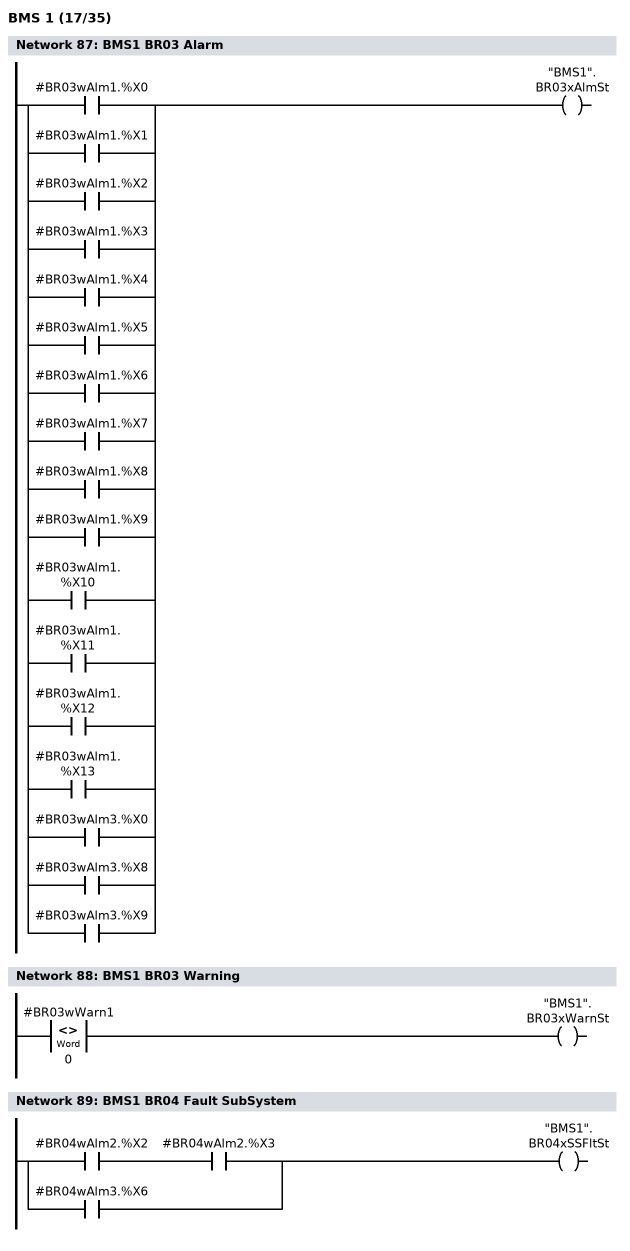
   RUNG wire#powerrail
      Contact( #BR03wAlm1.%X0 )
      wire#w1
      Coil( "BMS1".BR03xAlmSt )
   END_RUNG
   RUNG wire#powerrail
      Contact( #BR03wAlm1.%X1 )
   END_RUNG wire#w1
   RUNG wire#powerrail
      Contact( #BR03wAlm1.%X2 )
   END_RUNG wire#w1
   RUNG wire#powerrail
      Contact( #BR03wAlm1.%X3 )
   END_RUNG wire#w1
   RUNG wire#powerrail
      Contact( #BR03wAlm1.%X4 )
   END_RUNG wire#w1
   RUNG wire#powerrail
      Contact( #BR03wAlm1.%X5 )
   END_RUNG wire#w1
   RUNG wire#powerrail
      Contact( #BR03wAlm1.%X6 )
   END_RUNG wire#w1
   RUNG wire#powerrail
      Contact( #BR03wAlm1.%X7 )
   END_RUNG wire#w1
   RUNG wire#powerrail
      Contact( #BR03wAlm1.%X8 )
   END_RUNG wire#w1
   RUNG wire#powerrail
      Contact( #BR03wAlm1.%X9 )
   END_RUNG wire#w1
   RUNG wire#powerrail
      Contact( #BR03wAlm1.%X10 )
   END_RUNG wire#w1
   RUNG wire#powerrail
      Contact( #BR03wAlm1.%X11 )
   END_RUNG wire#w1
   RUNG wire#powerrail
      Contact( #BR03wAlm1.%X12 )
   END_RUNG wire#w1
   RUNG wire#powerrail
      Contact( #BR03wAlm1.%X13 )
   END_RUNG wire#w1
   RUNG wire#powerrail
      Contact( #BR03wAlm3.%X0 )
   END_RUNG wire#w1
   RUNG wire#powerrail
      Contact( #BR03wAlm3.%X8 )
   END_RUNG wire#w1
   RUNG wire#powerrail
      Contact( #BR03wAlm3.%X9 )
   END_RUNG wire#w1
   // the same network as SCL:
   "BMS1".BR03xAlmSt := #BR03wAlm1.%X0 OR #BR03wAlm1.%X1 OR #BR03wAlm1.%X2 OR #BR03wAlm1.%X3 OR #BR03wAlm1.%X4 OR #BR03wAlm1.%X5 OR #BR03wAlm1.%X6 OR #BR03wAlm1.%X7 OR #BR03wAlm1.%X8 OR #BR03wAlm1.%X9 OR #BR03wAlm1.%X10 OR #BR03wAlm1.%X11 OR #BR03wAlm1.%X12 OR #BR03wAlm1.%X13 OR #BR03wAlm3.%X0 OR #BR03wAlm3.%X8 OR #BR03wAlm3.%X9;
END_REGION

REGION Network 88: BMS1 BR03 Warning
   RUNG wire#powerrail
      { S7_Templates := "SrcType := Word" } NE_Contact(in1 := #BR03wWarn1, in2 := 0)
      Coil( "BMS1".BR03xWarnSt )
   END_RUNG
   // the same network as SCL:
   "BMS1".BR03xWarnSt := #BR03wWarn1 <> 0;
END_REGION

REGION Network 89: BMS1 BR04 Fault SubSystem
   RUNG wire#powerrail
      Contact( #BR04wAlm2.%X2 )
      Contact( #BR04wAlm2.%X3 )
      wire#w1
      Coil( "BMS1".BR04xSSFltSt )
   END_RUNG
   RUNG wire#powerrail
      Contact( #BR04wAlm3.%X6 )
   END_RUNG wire#w1
   // the same network as SCL:
   "BMS1".BR04xSSFltSt := (#BR04wAlm2.%X2 AND #BR04wAlm2.%X3) OR #BR04wAlm3.%X6;
END_REGION

REGION Network 90: BMS1 BR04 Fault
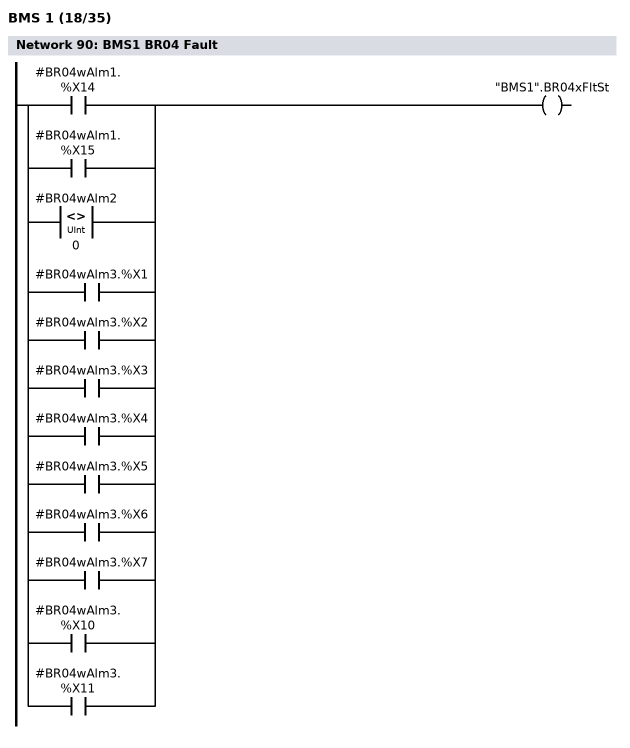
   RUNG wire#powerrail
      Contact( #BR04wAlm1.%X14 )
      wire#w1
      Coil( "BMS1".BR04xFltSt )
   END_RUNG
   RUNG wire#powerrail
      Contact( #BR04wAlm1.%X15 )
   END_RUNG wire#w1
   RUNG wire#powerrail
      { S7_Templates := "SrcType := UInt" } NE_Contact(in1 := #BR04wAlm2, in2 := 0)
   END_RUNG wire#w1
   RUNG wire#powerrail
      Contact( #BR04wAlm3.%X1 )
   END_RUNG wire#w1
   RUNG wire#powerrail
      Contact( #BR04wAlm3.%X2 )
   END_RUNG wire#w1
   RUNG wire#powerrail
      Contact( #BR04wAlm3.%X3 )
   END_RUNG wire#w1
   RUNG wire#powerrail
      Contact( #BR04wAlm3.%X4 )
   END_RUNG wire#w1
   RUNG wire#powerrail
      Contact( #BR04wAlm3.%X5 )
   END_RUNG wire#w1
   RUNG wire#powerrail
      Contact( #BR04wAlm3.%X6 )
   END_RUNG wire#w1
   RUNG wire#powerrail
      Contact( #BR04wAlm3.%X7 )
   END_RUNG wire#w1
   RUNG wire#powerrail
      Contact( #BR04wAlm3.%X10 )
   END_RUNG wire#w1
   RUNG wire#powerrail
      Contact( #BR04wAlm3.%X11 )
   END_RUNG wire#w1
   // the same network as SCL:
   "BMS1".BR04xFltSt := #BR04wAlm1.%X14 OR #BR04wAlm1.%X15 OR (#BR04wAlm2 <> 0) OR #BR04wAlm3.%X1 OR #BR04wAlm3.%X2 OR #BR04wAlm3.%X3 OR #BR04wAlm3.%X4 OR #BR04wAlm3.%X5 OR #BR04wAlm3.%X6 OR #BR04wAlm3.%X7 OR #BR04wAlm3.%X10 OR #BR04wAlm3.%X11;
END_REGION

REGION Network 91: BMS1 BR04 Alarm
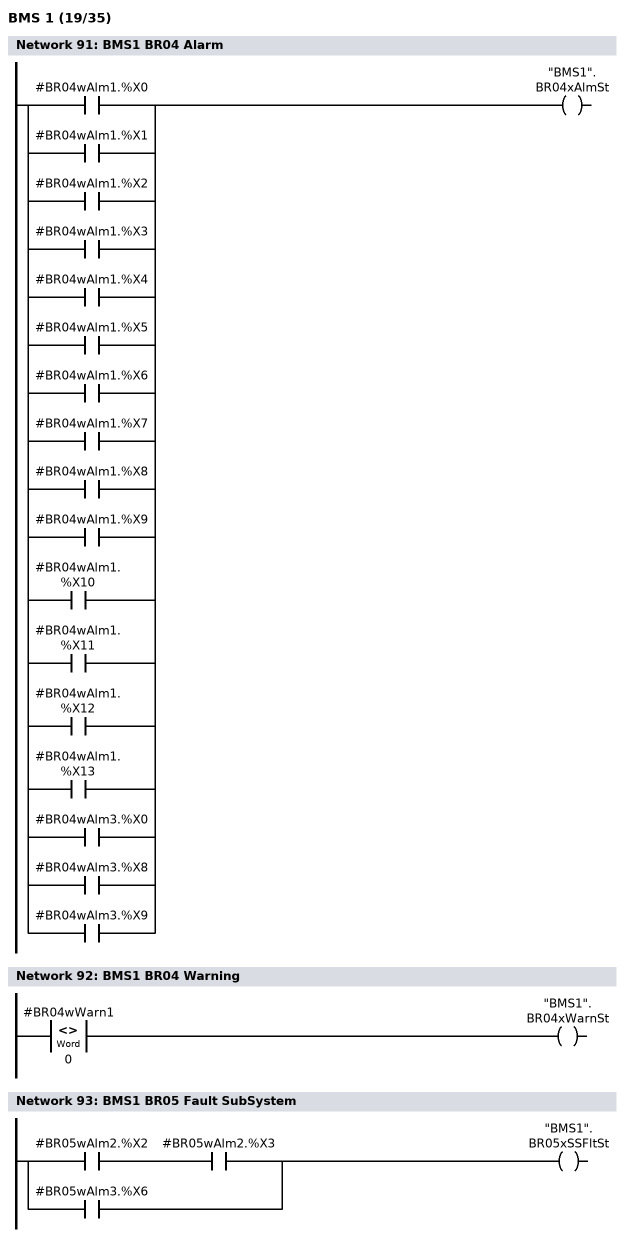
   RUNG wire#powerrail
      Contact( #BR04wAlm1.%X0 )
      wire#w1
      Coil( "BMS1".BR04xAlmSt )
   END_RUNG
   RUNG wire#powerrail
      Contact( #BR04wAlm1.%X1 )
   END_RUNG wire#w1
   RUNG wire#powerrail
      Contact( #BR04wAlm1.%X2 )
   END_RUNG wire#w1
   RUNG wire#powerrail
      Contact( #BR04wAlm1.%X3 )
   END_RUNG wire#w1
   RUNG wire#powerrail
      Contact( #BR04wAlm1.%X4 )
   END_RUNG wire#w1
   RUNG wire#powerrail
      Contact( #BR04wAlm1.%X5 )
   END_RUNG wire#w1
   RUNG wire#powerrail
      Contact( #BR04wAlm1.%X6 )
   END_RUNG wire#w1
   RUNG wire#powerrail
      Contact( #BR04wAlm1.%X7 )
   END_RUNG wire#w1
   RUNG wire#powerrail
      Contact( #BR04wAlm1.%X8 )
   END_RUNG wire#w1
   RUNG wire#powerrail
      Contact( #BR04wAlm1.%X9 )
   END_RUNG wire#w1
   RUNG wire#powerrail
      Contact( #BR04wAlm1.%X10 )
   END_RUNG wire#w1
   RUNG wire#powerrail
      Contact( #BR04wAlm1.%X11 )
   END_RUNG wire#w1
   RUNG wire#powerrail
      Contact( #BR04wAlm1.%X12 )
   END_RUNG wire#w1
   RUNG wire#powerrail
      Contact( #BR04wAlm1.%X13 )
   END_RUNG wire#w1
   RUNG wire#powerrail
      Contact( #BR04wAlm3.%X0 )
   END_RUNG wire#w1
   RUNG wire#powerrail
      Contact( #BR04wAlm3.%X8 )
   END_RUNG wire#w1
   RUNG wire#powerrail
      Contact( #BR04wAlm3.%X9 )
   END_RUNG wire#w1
   // the same network as SCL:
   "BMS1".BR04xAlmSt := #BR04wAlm1.%X0 OR #BR04wAlm1.%X1 OR #BR04wAlm1.%X2 OR #BR04wAlm1.%X3 OR #BR04wAlm1.%X4 OR #BR04wAlm1.%X5 OR #BR04wAlm1.%X6 OR #BR04wAlm1.%X7 OR #BR04wAlm1.%X8 OR #BR04wAlm1.%X9 OR #BR04wAlm1.%X10 OR #BR04wAlm1.%X11 OR #BR04wAlm1.%X12 OR #BR04wAlm1.%X13 OR #BR04wAlm3.%X0 OR #BR04wAlm3.%X8 OR #BR04wAlm3.%X9;
END_REGION

REGION Network 92: BMS1 BR04 Warning
   RUNG wire#powerrail
      { S7_Templates := "SrcType := Word" } NE_Contact(in1 := #BR04wWarn1, in2 := 0)
      Coil( "BMS1".BR04xWarnSt )
   END_RUNG
   // the same network as SCL:
   "BMS1".BR04xWarnSt := #BR04wWarn1 <> 0;
END_REGION

REGION Network 93: BMS1 BR05 Fault SubSystem
   RUNG wire#powerrail
      Contact( #BR05wAlm2.%X2 )
      Contact( #BR05wAlm2.%X3 )
      wire#w1
      Coil( "BMS1".BR05xSSFltSt )
   END_RUNG
   RUNG wire#powerrail
      Contact( #BR05wAlm3.%X6 )
   END_RUNG wire#w1
   // the same network as SCL:
   "BMS1".BR05xSSFltSt := (#BR05wAlm2.%X2 AND #BR05wAlm2.%X3) OR #BR05wAlm3.%X6;
END_REGION

REGION Network 94: BMS1 BR05 Fault
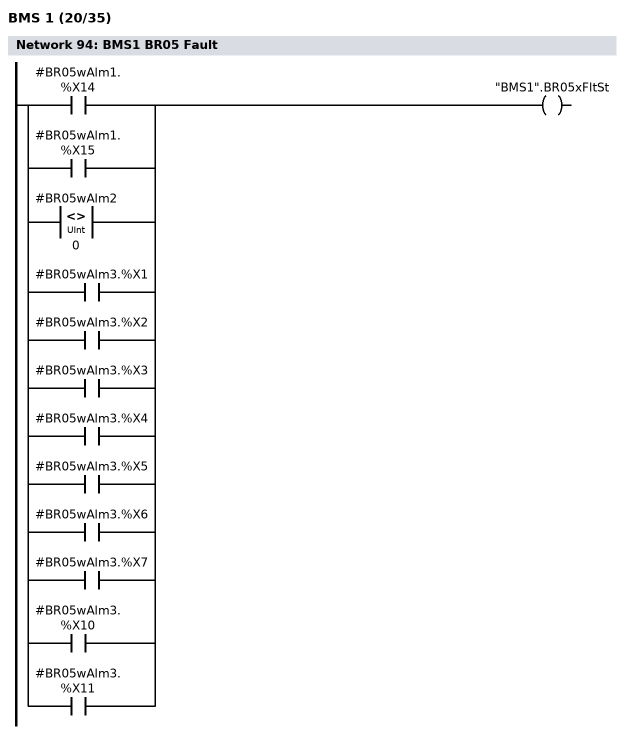
   RUNG wire#powerrail
      Contact( #BR05wAlm1.%X14 )
      wire#w1
      Coil( "BMS1".BR05xFltSt )
   END_RUNG
   RUNG wire#powerrail
      Contact( #BR05wAlm1.%X15 )
   END_RUNG wire#w1
   RUNG wire#powerrail
      { S7_Templates := "SrcType := UInt" } NE_Contact(in1 := #BR05wAlm2, in2 := 0)
   END_RUNG wire#w1
   RUNG wire#powerrail
      Contact( #BR05wAlm3.%X1 )
   END_RUNG wire#w1
   RUNG wire#powerrail
      Contact( #BR05wAlm3.%X2 )
   END_RUNG wire#w1
   RUNG wire#powerrail
      Contact( #BR05wAlm3.%X3 )
   END_RUNG wire#w1
   RUNG wire#powerrail
      Contact( #BR05wAlm3.%X4 )
   END_RUNG wire#w1
   RUNG wire#powerrail
      Contact( #BR05wAlm3.%X5 )
   END_RUNG wire#w1
   RUNG wire#powerrail
      Contact( #BR05wAlm3.%X6 )
   END_RUNG wire#w1
   RUNG wire#powerrail
      Contact( #BR05wAlm3.%X7 )
   END_RUNG wire#w1
   RUNG wire#powerrail
      Contact( #BR05wAlm3.%X10 )
   END_RUNG wire#w1
   RUNG wire#powerrail
      Contact( #BR05wAlm3.%X11 )
   END_RUNG wire#w1
   // the same network as SCL:
   "BMS1".BR05xFltSt := #BR05wAlm1.%X14 OR #BR05wAlm1.%X15 OR (#BR05wAlm2 <> 0) OR #BR05wAlm3.%X1 OR #BR05wAlm3.%X2 OR #BR05wAlm3.%X3 OR #BR05wAlm3.%X4 OR #BR05wAlm3.%X5 OR #BR05wAlm3.%X6 OR #BR05wAlm3.%X7 OR #BR05wAlm3.%X10 OR #BR05wAlm3.%X11;
END_REGION

REGION Network 95: BMS1 BR05 Alarm
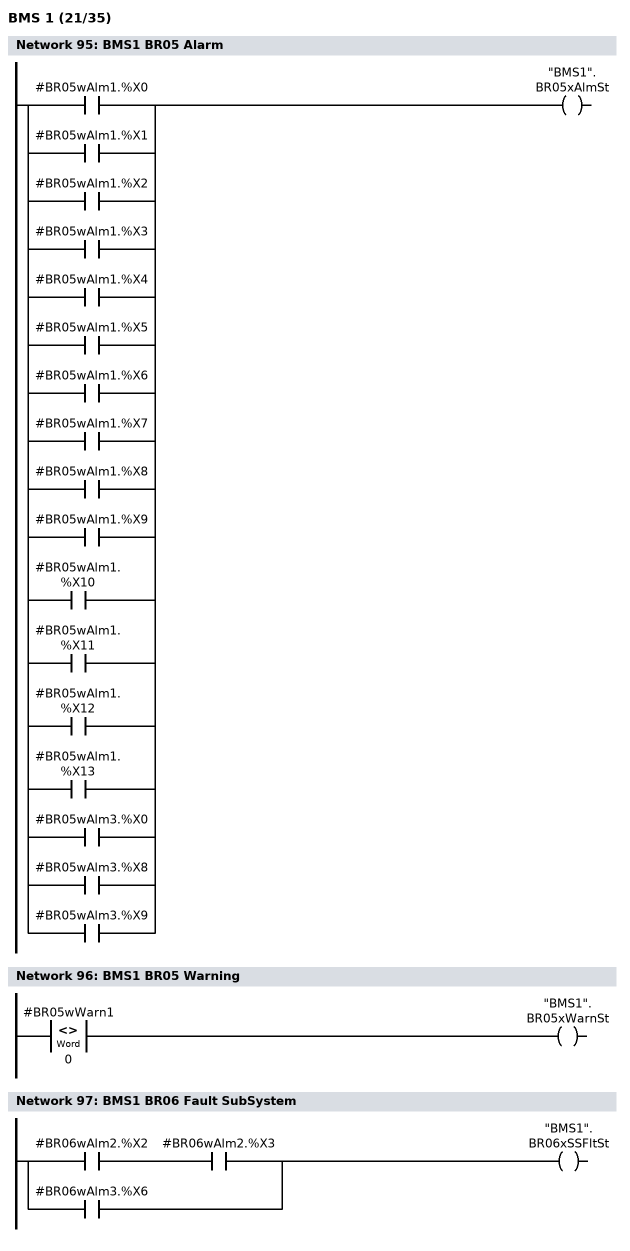
   RUNG wire#powerrail
      Contact( #BR05wAlm1.%X0 )
      wire#w1
      Coil( "BMS1".BR05xAlmSt )
   END_RUNG
   RUNG wire#powerrail
      Contact( #BR05wAlm1.%X1 )
   END_RUNG wire#w1
   RUNG wire#powerrail
      Contact( #BR05wAlm1.%X2 )
   END_RUNG wire#w1
   RUNG wire#powerrail
      Contact( #BR05wAlm1.%X3 )
   END_RUNG wire#w1
   RUNG wire#powerrail
      Contact( #BR05wAlm1.%X4 )
   END_RUNG wire#w1
   RUNG wire#powerrail
      Contact( #BR05wAlm1.%X5 )
   END_RUNG wire#w1
   RUNG wire#powerrail
      Contact( #BR05wAlm1.%X6 )
   END_RUNG wire#w1
   RUNG wire#powerrail
      Contact( #BR05wAlm1.%X7 )
   END_RUNG wire#w1
   RUNG wire#powerrail
      Contact( #BR05wAlm1.%X8 )
   END_RUNG wire#w1
   RUNG wire#powerrail
      Contact( #BR05wAlm1.%X9 )
   END_RUNG wire#w1
   RUNG wire#powerrail
      Contact( #BR05wAlm1.%X10 )
   END_RUNG wire#w1
   RUNG wire#powerrail
      Contact( #BR05wAlm1.%X11 )
   END_RUNG wire#w1
   RUNG wire#powerrail
      Contact( #BR05wAlm1.%X12 )
   END_RUNG wire#w1
   RUNG wire#powerrail
      Contact( #BR05wAlm1.%X13 )
   END_RUNG wire#w1
   RUNG wire#powerrail
      Contact( #BR05wAlm3.%X0 )
   END_RUNG wire#w1
   RUNG wire#powerrail
      Contact( #BR05wAlm3.%X8 )
   END_RUNG wire#w1
   RUNG wire#powerrail
      Contact( #BR05wAlm3.%X9 )
   END_RUNG wire#w1
   // the same network as SCL:
   "BMS1".BR05xAlmSt := #BR05wAlm1.%X0 OR #BR05wAlm1.%X1 OR #BR05wAlm1.%X2 OR #BR05wAlm1.%X3 OR #BR05wAlm1.%X4 OR #BR05wAlm1.%X5 OR #BR05wAlm1.%X6 OR #BR05wAlm1.%X7 OR #BR05wAlm1.%X8 OR #BR05wAlm1.%X9 OR #BR05wAlm1.%X10 OR #BR05wAlm1.%X11 OR #BR05wAlm1.%X12 OR #BR05wAlm1.%X13 OR #BR05wAlm3.%X0 OR #BR05wAlm3.%X8 OR #BR05wAlm3.%X9;
END_REGION

REGION Network 96: BMS1 BR05 Warning
   RUNG wire#powerrail
      { S7_Templates := "SrcType := Word" } NE_Contact(in1 := #BR05wWarn1, in2 := 0)
      Coil( "BMS1".BR05xWarnSt )
   END_RUNG
   // the same network as SCL:
   "BMS1".BR05xWarnSt := #BR05wWarn1 <> 0;
END_REGION

REGION Network 97: BMS1 BR06 Fault SubSystem
   RUNG wire#powerrail
      Contact( #BR06wAlm2.%X2 )
      Contact( #BR06wAlm2.%X3 )
      wire#w1
      Coil( "BMS1".BR06xSSFltSt )
   END_RUNG
   RUNG wire#powerrail
      Contact( #BR06wAlm3.%X6 )
   END_RUNG wire#w1
   // the same network as SCL:
   "BMS1".BR06xSSFltSt := (#BR06wAlm2.%X2 AND #BR06wAlm2.%X3) OR #BR06wAlm3.%X6;
END_REGION

REGION Network 98: BMS1 BR06 Fault
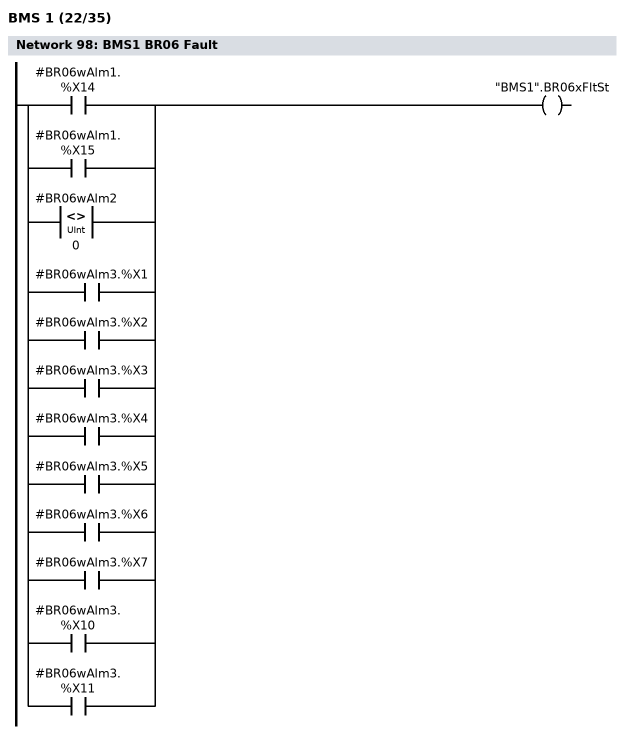
   RUNG wire#powerrail
      Contact( #BR06wAlm1.%X14 )
      wire#w1
      Coil( "BMS1".BR06xFltSt )
   END_RUNG
   RUNG wire#powerrail
      Contact( #BR06wAlm1.%X15 )
   END_RUNG wire#w1
   RUNG wire#powerrail
      { S7_Templates := "SrcType := UInt" } NE_Contact(in1 := #BR06wAlm2, in2 := 0)
   END_RUNG wire#w1
   RUNG wire#powerrail
      Contact( #BR06wAlm3.%X1 )
   END_RUNG wire#w1
   RUNG wire#powerrail
      Contact( #BR06wAlm3.%X2 )
   END_RUNG wire#w1
   RUNG wire#powerrail
      Contact( #BR06wAlm3.%X3 )
   END_RUNG wire#w1
   RUNG wire#powerrail
      Contact( #BR06wAlm3.%X4 )
   END_RUNG wire#w1
   RUNG wire#powerrail
      Contact( #BR06wAlm3.%X5 )
   END_RUNG wire#w1
   RUNG wire#powerrail
      Contact( #BR06wAlm3.%X6 )
   END_RUNG wire#w1
   RUNG wire#powerrail
      Contact( #BR06wAlm3.%X7 )
   END_RUNG wire#w1
   RUNG wire#powerrail
      Contact( #BR06wAlm3.%X10 )
   END_RUNG wire#w1
   RUNG wire#powerrail
      Contact( #BR06wAlm3.%X11 )
   END_RUNG wire#w1
   // the same network as SCL:
   "BMS1".BR06xFltSt := #BR06wAlm1.%X14 OR #BR06wAlm1.%X15 OR (#BR06wAlm2 <> 0) OR #BR06wAlm3.%X1 OR #BR06wAlm3.%X2 OR #BR06wAlm3.%X3 OR #BR06wAlm3.%X4 OR #BR06wAlm3.%X5 OR #BR06wAlm3.%X6 OR #BR06wAlm3.%X7 OR #BR06wAlm3.%X10 OR #BR06wAlm3.%X11;
END_REGION

REGION Network 99: BMS1 BR06 Alarm
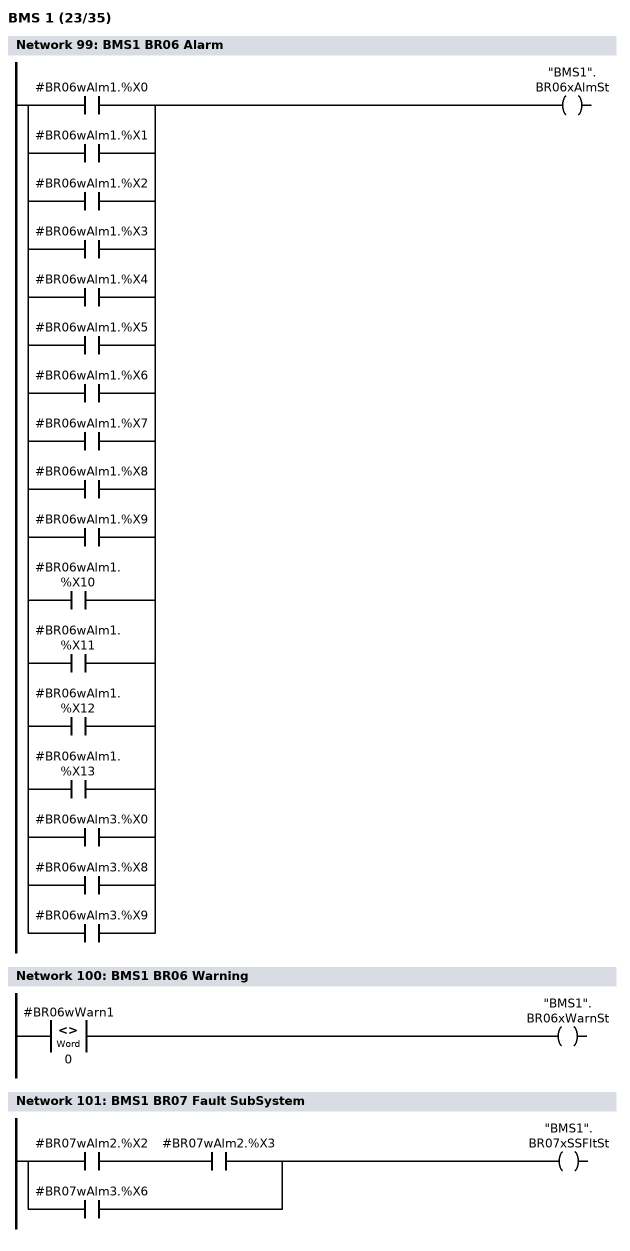
   RUNG wire#powerrail
      Contact( #BR06wAlm1.%X0 )
      wire#w1
      Coil( "BMS1".BR06xAlmSt )
   END_RUNG
   RUNG wire#powerrail
      Contact( #BR06wAlm1.%X1 )
   END_RUNG wire#w1
   RUNG wire#powerrail
      Contact( #BR06wAlm1.%X2 )
   END_RUNG wire#w1
   RUNG wire#powerrail
      Contact( #BR06wAlm1.%X3 )
   END_RUNG wire#w1
   RUNG wire#powerrail
      Contact( #BR06wAlm1.%X4 )
   END_RUNG wire#w1
   RUNG wire#powerrail
      Contact( #BR06wAlm1.%X5 )
   END_RUNG wire#w1
   RUNG wire#powerrail
      Contact( #BR06wAlm1.%X6 )
   END_RUNG wire#w1
   RUNG wire#powerrail
      Contact( #BR06wAlm1.%X7 )
   END_RUNG wire#w1
   RUNG wire#powerrail
      Contact( #BR06wAlm1.%X8 )
   END_RUNG wire#w1
   RUNG wire#powerrail
      Contact( #BR06wAlm1.%X9 )
   END_RUNG wire#w1
   RUNG wire#powerrail
      Contact( #BR06wAlm1.%X10 )
   END_RUNG wire#w1
   RUNG wire#powerrail
      Contact( #BR06wAlm1.%X11 )
   END_RUNG wire#w1
   RUNG wire#powerrail
      Contact( #BR06wAlm1.%X12 )
   END_RUNG wire#w1
   RUNG wire#powerrail
      Contact( #BR06wAlm1.%X13 )
   END_RUNG wire#w1
   RUNG wire#powerrail
      Contact( #BR06wAlm3.%X0 )
   END_RUNG wire#w1
   RUNG wire#powerrail
      Contact( #BR06wAlm3.%X8 )
   END_RUNG wire#w1
   RUNG wire#powerrail
      Contact( #BR06wAlm3.%X9 )
   END_RUNG wire#w1
   // the same network as SCL:
   "BMS1".BR06xAlmSt := #BR06wAlm1.%X0 OR #BR06wAlm1.%X1 OR #BR06wAlm1.%X2 OR #BR06wAlm1.%X3 OR #BR06wAlm1.%X4 OR #BR06wAlm1.%X5 OR #BR06wAlm1.%X6 OR #BR06wAlm1.%X7 OR #BR06wAlm1.%X8 OR #BR06wAlm1.%X9 OR #BR06wAlm1.%X10 OR #BR06wAlm1.%X11 OR #BR06wAlm1.%X12 OR #BR06wAlm1.%X13 OR #BR06wAlm3.%X0 OR #BR06wAlm3.%X8 OR #BR06wAlm3.%X9;
END_REGION

REGION Network 100: BMS1 BR06 Warning
   RUNG wire#powerrail
      { S7_Templates := "SrcType := Word" } NE_Contact(in1 := #BR06wWarn1, in2 := 0)
      Coil( "BMS1".BR06xWarnSt )
   END_RUNG
   // the same network as SCL:
   "BMS1".BR06xWarnSt := #BR06wWarn1 <> 0;
END_REGION

REGION Network 101: BMS1 BR07 Fault SubSystem
   RUNG wire#powerrail
      Contact( #BR07wAlm2.%X2 )
      Contact( #BR07wAlm2.%X3 )
      wire#w1
      Coil( "BMS1".BR07xSSFltSt )
   END_RUNG
   RUNG wire#powerrail
      Contact( #BR07wAlm3.%X6 )
   END_RUNG wire#w1
   // the same network as SCL:
   "BMS1".BR07xSSFltSt := (#BR07wAlm2.%X2 AND #BR07wAlm2.%X3) OR #BR07wAlm3.%X6;
END_REGION

REGION Network 102: BMS1 BR07 Fault
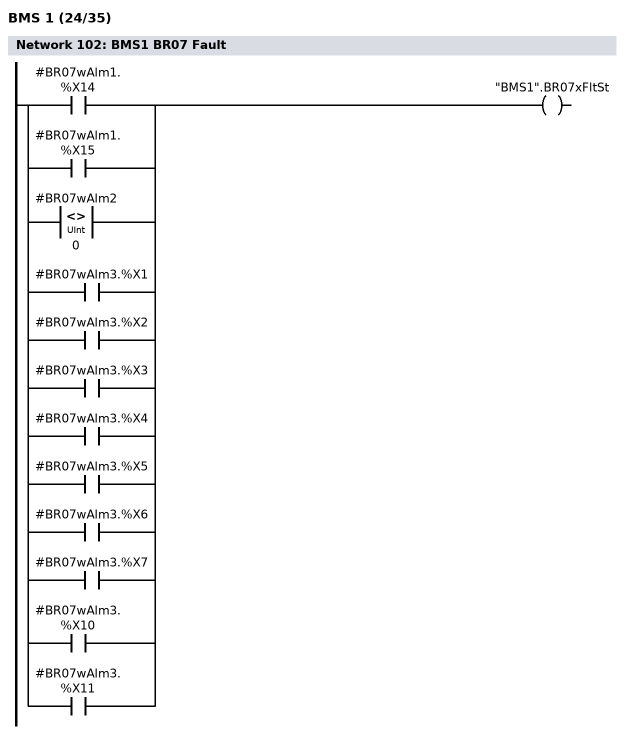
   RUNG wire#powerrail
      Contact( #BR07wAlm1.%X14 )
      wire#w1
      Coil( "BMS1".BR07xFltSt )
   END_RUNG
   RUNG wire#powerrail
      Contact( #BR07wAlm1.%X15 )
   END_RUNG wire#w1
   RUNG wire#powerrail
      { S7_Templates := "SrcType := UInt" } NE_Contact(in1 := #BR07wAlm2, in2 := 0)
   END_RUNG wire#w1
   RUNG wire#powerrail
      Contact( #BR07wAlm3.%X1 )
   END_RUNG wire#w1
   RUNG wire#powerrail
      Contact( #BR07wAlm3.%X2 )
   END_RUNG wire#w1
   RUNG wire#powerrail
      Contact( #BR07wAlm3.%X3 )
   END_RUNG wire#w1
   RUNG wire#powerrail
      Contact( #BR07wAlm3.%X4 )
   END_RUNG wire#w1
   RUNG wire#powerrail
      Contact( #BR07wAlm3.%X5 )
   END_RUNG wire#w1
   RUNG wire#powerrail
      Contact( #BR07wAlm3.%X6 )
   END_RUNG wire#w1
   RUNG wire#powerrail
      Contact( #BR07wAlm3.%X7 )
   END_RUNG wire#w1
   RUNG wire#powerrail
      Contact( #BR07wAlm3.%X10 )
   END_RUNG wire#w1
   RUNG wire#powerrail
      Contact( #BR07wAlm3.%X11 )
   END_RUNG wire#w1
   // the same network as SCL:
   "BMS1".BR07xFltSt := #BR07wAlm1.%X14 OR #BR07wAlm1.%X15 OR (#BR07wAlm2 <> 0) OR #BR07wAlm3.%X1 OR #BR07wAlm3.%X2 OR #BR07wAlm3.%X3 OR #BR07wAlm3.%X4 OR #BR07wAlm3.%X5 OR #BR07wAlm3.%X6 OR #BR07wAlm3.%X7 OR #BR07wAlm3.%X10 OR #BR07wAlm3.%X11;
END_REGION

REGION Network 103: BMS1 BR07 Alarm
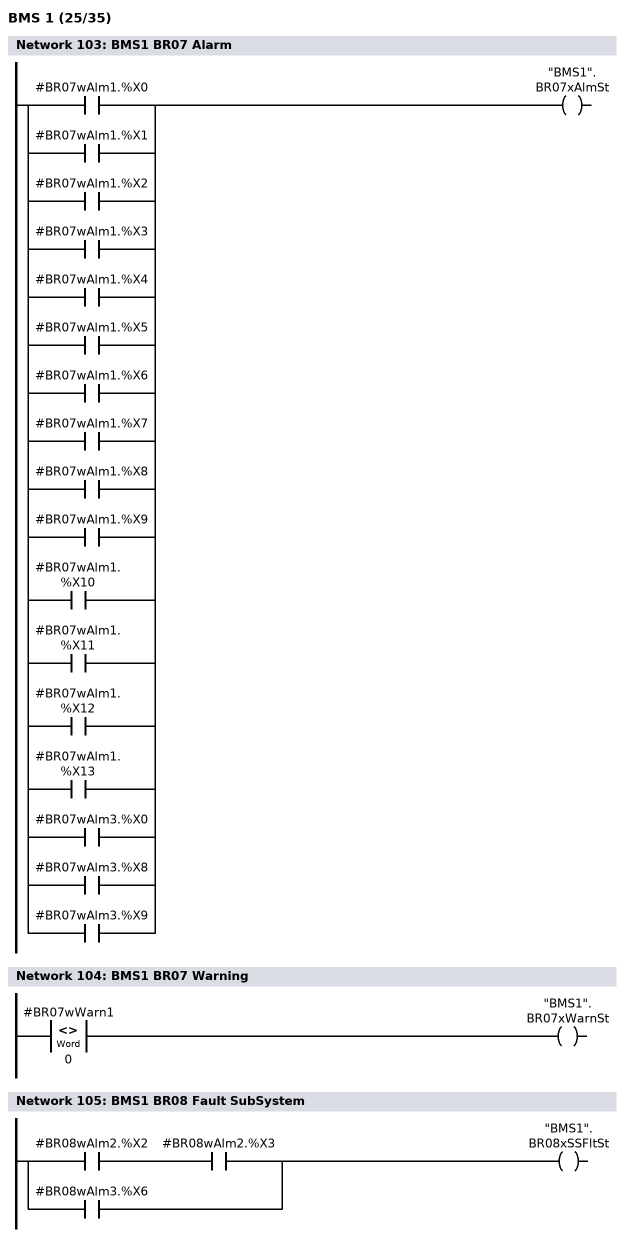
   RUNG wire#powerrail
      Contact( #BR07wAlm1.%X0 )
      wire#w1
      Coil( "BMS1".BR07xAlmSt )
   END_RUNG
   RUNG wire#powerrail
      Contact( #BR07wAlm1.%X1 )
   END_RUNG wire#w1
   RUNG wire#powerrail
      Contact( #BR07wAlm1.%X2 )
   END_RUNG wire#w1
   RUNG wire#powerrail
      Contact( #BR07wAlm1.%X3 )
   END_RUNG wire#w1
   RUNG wire#powerrail
      Contact( #BR07wAlm1.%X4 )
   END_RUNG wire#w1
   RUNG wire#powerrail
      Contact( #BR07wAlm1.%X5 )
   END_RUNG wire#w1
   RUNG wire#powerrail
      Contact( #BR07wAlm1.%X6 )
   END_RUNG wire#w1
   RUNG wire#powerrail
      Contact( #BR07wAlm1.%X7 )
   END_RUNG wire#w1
   RUNG wire#powerrail
      Contact( #BR07wAlm1.%X8 )
   END_RUNG wire#w1
   RUNG wire#powerrail
      Contact( #BR07wAlm1.%X9 )
   END_RUNG wire#w1
   RUNG wire#powerrail
      Contact( #BR07wAlm1.%X10 )
   END_RUNG wire#w1
   RUNG wire#powerrail
      Contact( #BR07wAlm1.%X11 )
   END_RUNG wire#w1
   RUNG wire#powerrail
      Contact( #BR07wAlm1.%X12 )
   END_RUNG wire#w1
   RUNG wire#powerrail
      Contact( #BR07wAlm1.%X13 )
   END_RUNG wire#w1
   RUNG wire#powerrail
      Contact( #BR07wAlm3.%X0 )
   END_RUNG wire#w1
   RUNG wire#powerrail
      Contact( #BR07wAlm3.%X8 )
   END_RUNG wire#w1
   RUNG wire#powerrail
      Contact( #BR07wAlm3.%X9 )
   END_RUNG wire#w1
   // the same network as SCL:
   "BMS1".BR07xAlmSt := #BR07wAlm1.%X0 OR #BR07wAlm1.%X1 OR #BR07wAlm1.%X2 OR #BR07wAlm1.%X3 OR #BR07wAlm1.%X4 OR #BR07wAlm1.%X5 OR #BR07wAlm1.%X6 OR #BR07wAlm1.%X7 OR #BR07wAlm1.%X8 OR #BR07wAlm1.%X9 OR #BR07wAlm1.%X10 OR #BR07wAlm1.%X11 OR #BR07wAlm1.%X12 OR #BR07wAlm1.%X13 OR #BR07wAlm3.%X0 OR #BR07wAlm3.%X8 OR #BR07wAlm3.%X9;
END_REGION

REGION Network 104: BMS1 BR07 Warning
   RUNG wire#powerrail
      { S7_Templates := "SrcType := Word" } NE_Contact(in1 := #BR07wWarn1, in2 := 0)
      Coil( "BMS1".BR07xWarnSt )
   END_RUNG
   // the same network as SCL:
   "BMS1".BR07xWarnSt := #BR07wWarn1 <> 0;
END_REGION

REGION Network 105: BMS1 BR08 Fault SubSystem
   RUNG wire#powerrail
      Contact( #BR08wAlm2.%X2 )
      Contact( #BR08wAlm2.%X3 )
      wire#w1
      Coil( "BMS1".BR08xSSFltSt )
   END_RUNG
   RUNG wire#powerrail
      Contact( #BR08wAlm3.%X6 )
   END_RUNG wire#w1
   // the same network as SCL:
   "BMS1".BR08xSSFltSt := (#BR08wAlm2.%X2 AND #BR08wAlm2.%X3) OR #BR08wAlm3.%X6;
END_REGION

REGION Network 106: BMS1 BR08 Fault
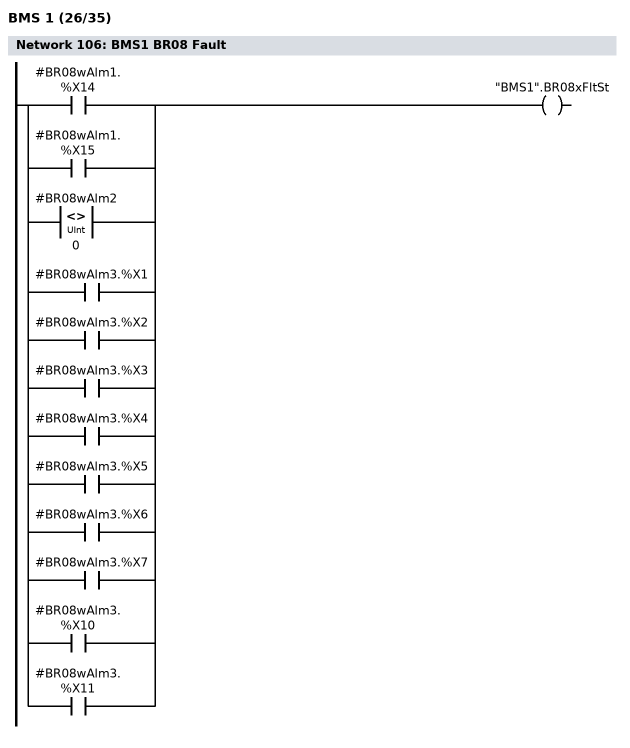
   RUNG wire#powerrail
      Contact( #BR08wAlm1.%X14 )
      wire#w1
      Coil( "BMS1".BR08xFltSt )
   END_RUNG
   RUNG wire#powerrail
      Contact( #BR08wAlm1.%X15 )
   END_RUNG wire#w1
   RUNG wire#powerrail
      { S7_Templates := "SrcType := UInt" } NE_Contact(in1 := #BR08wAlm2, in2 := 0)
   END_RUNG wire#w1
   RUNG wire#powerrail
      Contact( #BR08wAlm3.%X1 )
   END_RUNG wire#w1
   RUNG wire#powerrail
      Contact( #BR08wAlm3.%X2 )
   END_RUNG wire#w1
   RUNG wire#powerrail
      Contact( #BR08wAlm3.%X3 )
   END_RUNG wire#w1
   RUNG wire#powerrail
      Contact( #BR08wAlm3.%X4 )
   END_RUNG wire#w1
   RUNG wire#powerrail
      Contact( #BR08wAlm3.%X5 )
   END_RUNG wire#w1
   RUNG wire#powerrail
      Contact( #BR08wAlm3.%X6 )
   END_RUNG wire#w1
   RUNG wire#powerrail
      Contact( #BR08wAlm3.%X7 )
   END_RUNG wire#w1
   RUNG wire#powerrail
      Contact( #BR08wAlm3.%X10 )
   END_RUNG wire#w1
   RUNG wire#powerrail
      Contact( #BR08wAlm3.%X11 )
   END_RUNG wire#w1
   // the same network as SCL:
   "BMS1".BR08xFltSt := #BR08wAlm1.%X14 OR #BR08wAlm1.%X15 OR (#BR08wAlm2 <> 0) OR #BR08wAlm3.%X1 OR #BR08wAlm3.%X2 OR #BR08wAlm3.%X3 OR #BR08wAlm3.%X4 OR #BR08wAlm3.%X5 OR #BR08wAlm3.%X6 OR #BR08wAlm3.%X7 OR #BR08wAlm3.%X10 OR #BR08wAlm3.%X11;
END_REGION

REGION Network 107: BMS1 BR08 Alarm
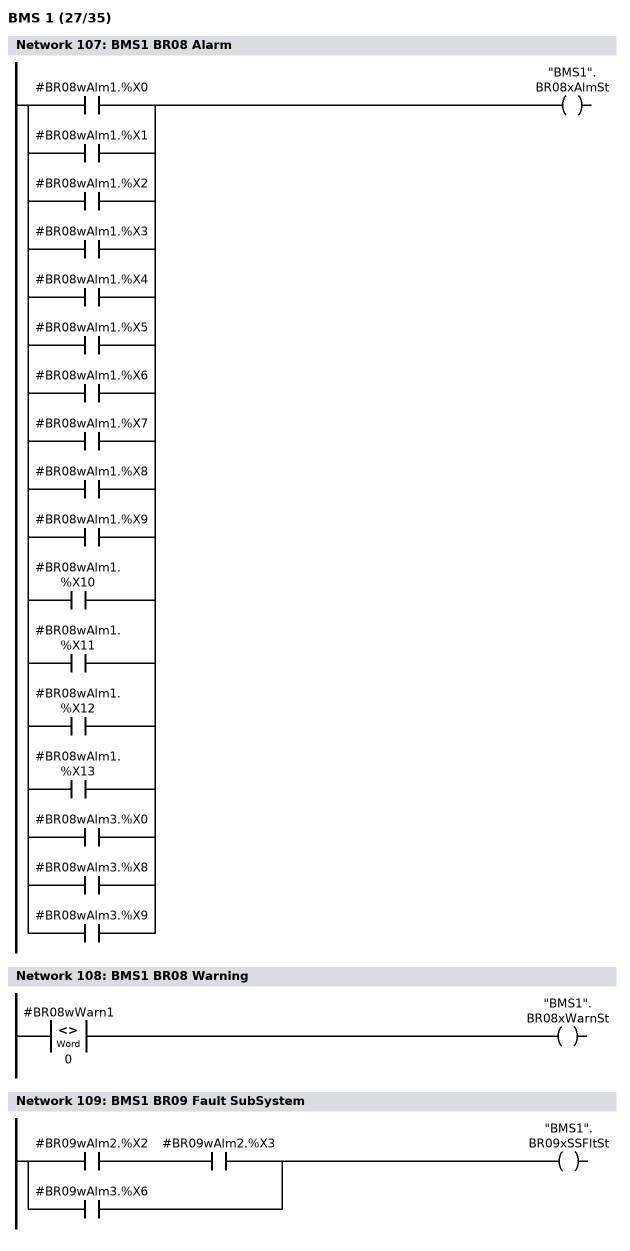
   RUNG wire#powerrail
      Contact( #BR08wAlm1.%X0 )
      wire#w1
      Coil( "BMS1".BR08xAlmSt )
   END_RUNG
   RUNG wire#powerrail
      Contact( #BR08wAlm1.%X1 )
   END_RUNG wire#w1
   RUNG wire#powerrail
      Contact( #BR08wAlm1.%X2 )
   END_RUNG wire#w1
   RUNG wire#powerrail
      Contact( #BR08wAlm1.%X3 )
   END_RUNG wire#w1
   RUNG wire#powerrail
      Contact( #BR08wAlm1.%X4 )
   END_RUNG wire#w1
   RUNG wire#powerrail
      Contact( #BR08wAlm1.%X5 )
   END_RUNG wire#w1
   RUNG wire#powerrail
      Contact( #BR08wAlm1.%X6 )
   END_RUNG wire#w1
   RUNG wire#powerrail
      Contact( #BR08wAlm1.%X7 )
   END_RUNG wire#w1
   RUNG wire#powerrail
      Contact( #BR08wAlm1.%X8 )
   END_RUNG wire#w1
   RUNG wire#powerrail
      Contact( #BR08wAlm1.%X9 )
   END_RUNG wire#w1
   RUNG wire#powerrail
      Contact( #BR08wAlm1.%X10 )
   END_RUNG wire#w1
   RUNG wire#powerrail
      Contact( #BR08wAlm1.%X11 )
   END_RUNG wire#w1
   RUNG wire#powerrail
      Contact( #BR08wAlm1.%X12 )
   END_RUNG wire#w1
   RUNG wire#powerrail
      Contact( #BR08wAlm1.%X13 )
   END_RUNG wire#w1
   RUNG wire#powerrail
      Contact( #BR08wAlm3.%X0 )
   END_RUNG wire#w1
   RUNG wire#powerrail
      Contact( #BR08wAlm3.%X8 )
   END_RUNG wire#w1
   RUNG wire#powerrail
      Contact( #BR08wAlm3.%X9 )
   END_RUNG wire#w1
   // the same network as SCL:
   "BMS1".BR08xAlmSt := #BR08wAlm1.%X0 OR #BR08wAlm1.%X1 OR #BR08wAlm1.%X2 OR #BR08wAlm1.%X3 OR #BR08wAlm1.%X4 OR #BR08wAlm1.%X5 OR #BR08wAlm1.%X6 OR #BR08wAlm1.%X7 OR #BR08wAlm1.%X8 OR #BR08wAlm1.%X9 OR #BR08wAlm1.%X10 OR #BR08wAlm1.%X11 OR #BR08wAlm1.%X12 OR #BR08wAlm1.%X13 OR #BR08wAlm3.%X0 OR #BR08wAlm3.%X8 OR #BR08wAlm3.%X9;
END_REGION

REGION Network 108: BMS1 BR08 Warning
   RUNG wire#powerrail
      { S7_Templates := "SrcType := Word" } NE_Contact(in1 := #BR08wWarn1, in2 := 0)
      Coil( "BMS1".BR08xWarnSt )
   END_RUNG
   // the same network as SCL:
   "BMS1".BR08xWarnSt := #BR08wWarn1 <> 0;
END_REGION

REGION Network 109: BMS1 BR09 Fault SubSystem
   RUNG wire#powerrail
      Contact( #BR09wAlm2.%X2 )
      Contact( #BR09wAlm2.%X3 )
      wire#w1
      Coil( "BMS1".BR09xSSFltSt )
   END_RUNG
   RUNG wire#powerrail
      Contact( #BR09wAlm3.%X6 )
   END_RUNG wire#w1
   // the same network as SCL:
   "BMS1".BR09xSSFltSt := (#BR09wAlm2.%X2 AND #BR09wAlm2.%X3) OR #BR09wAlm3.%X6;
END_REGION

REGION Network 110: BMS1 BR09 Fault
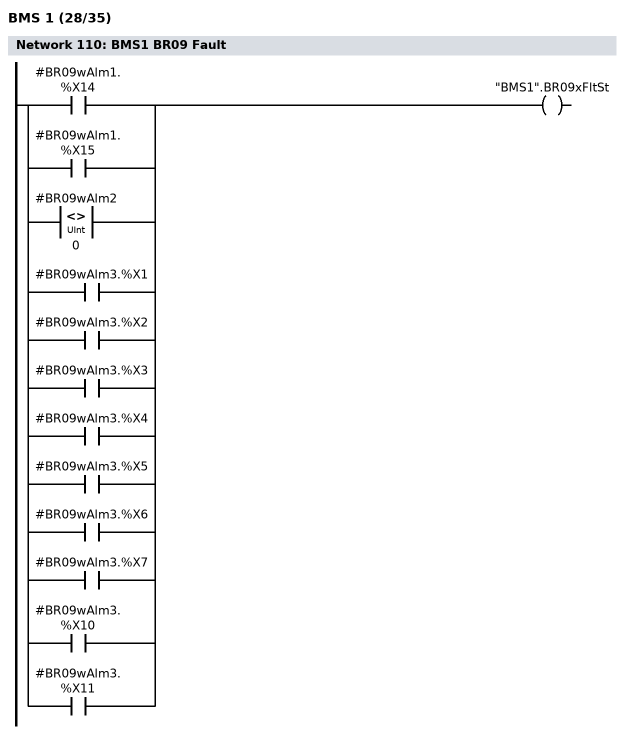
   RUNG wire#powerrail
      Contact( #BR09wAlm1.%X14 )
      wire#w1
      Coil( "BMS1".BR09xFltSt )
   END_RUNG
   RUNG wire#powerrail
      Contact( #BR09wAlm1.%X15 )
   END_RUNG wire#w1
   RUNG wire#powerrail
      { S7_Templates := "SrcType := UInt" } NE_Contact(in1 := #BR09wAlm2, in2 := 0)
   END_RUNG wire#w1
   RUNG wire#powerrail
      Contact( #BR09wAlm3.%X1 )
   END_RUNG wire#w1
   RUNG wire#powerrail
      Contact( #BR09wAlm3.%X2 )
   END_RUNG wire#w1
   RUNG wire#powerrail
      Contact( #BR09wAlm3.%X3 )
   END_RUNG wire#w1
   RUNG wire#powerrail
      Contact( #BR09wAlm3.%X4 )
   END_RUNG wire#w1
   RUNG wire#powerrail
      Contact( #BR09wAlm3.%X5 )
   END_RUNG wire#w1
   RUNG wire#powerrail
      Contact( #BR09wAlm3.%X6 )
   END_RUNG wire#w1
   RUNG wire#powerrail
      Contact( #BR09wAlm3.%X7 )
   END_RUNG wire#w1
   RUNG wire#powerrail
      Contact( #BR09wAlm3.%X10 )
   END_RUNG wire#w1
   RUNG wire#powerrail
      Contact( #BR09wAlm3.%X11 )
   END_RUNG wire#w1
   // the same network as SCL:
   "BMS1".BR09xFltSt := #BR09wAlm1.%X14 OR #BR09wAlm1.%X15 OR (#BR09wAlm2 <> 0) OR #BR09wAlm3.%X1 OR #BR09wAlm3.%X2 OR #BR09wAlm3.%X3 OR #BR09wAlm3.%X4 OR #BR09wAlm3.%X5 OR #BR09wAlm3.%X6 OR #BR09wAlm3.%X7 OR #BR09wAlm3.%X10 OR #BR09wAlm3.%X11;
END_REGION

REGION Network 111: BMS1 BR09 Alarm
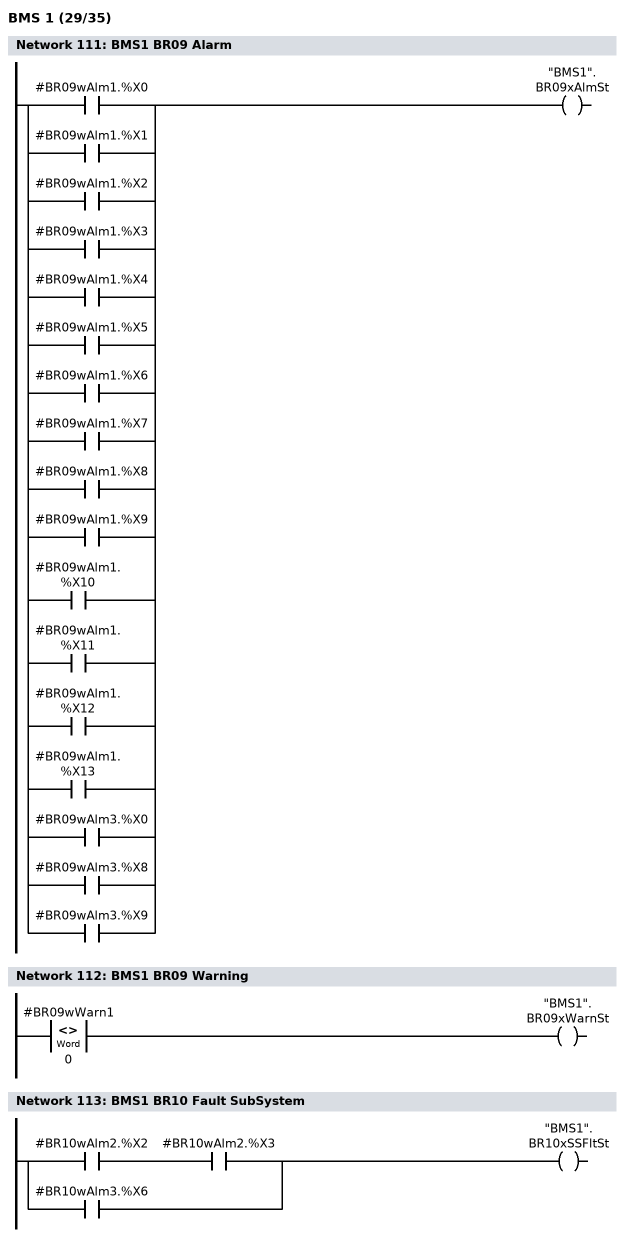
   RUNG wire#powerrail
      Contact( #BR09wAlm1.%X0 )
      wire#w1
      Coil( "BMS1".BR09xAlmSt )
   END_RUNG
   RUNG wire#powerrail
      Contact( #BR09wAlm1.%X1 )
   END_RUNG wire#w1
   RUNG wire#powerrail
      Contact( #BR09wAlm1.%X2 )
   END_RUNG wire#w1
   RUNG wire#powerrail
      Contact( #BR09wAlm1.%X3 )
   END_RUNG wire#w1
   RUNG wire#powerrail
      Contact( #BR09wAlm1.%X4 )
   END_RUNG wire#w1
   RUNG wire#powerrail
      Contact( #BR09wAlm1.%X5 )
   END_RUNG wire#w1
   RUNG wire#powerrail
      Contact( #BR09wAlm1.%X6 )
   END_RUNG wire#w1
   RUNG wire#powerrail
      Contact( #BR09wAlm1.%X7 )
   END_RUNG wire#w1
   RUNG wire#powerrail
      Contact( #BR09wAlm1.%X8 )
   END_RUNG wire#w1
   RUNG wire#powerrail
      Contact( #BR09wAlm1.%X9 )
   END_RUNG wire#w1
   RUNG wire#powerrail
      Contact( #BR09wAlm1.%X10 )
   END_RUNG wire#w1
   RUNG wire#powerrail
      Contact( #BR09wAlm1.%X11 )
   END_RUNG wire#w1
   RUNG wire#powerrail
      Contact( #BR09wAlm1.%X12 )
   END_RUNG wire#w1
   RUNG wire#powerrail
      Contact( #BR09wAlm1.%X13 )
   END_RUNG wire#w1
   RUNG wire#powerrail
      Contact( #BR09wAlm3.%X0 )
   END_RUNG wire#w1
   RUNG wire#powerrail
      Contact( #BR09wAlm3.%X8 )
   END_RUNG wire#w1
   RUNG wire#powerrail
      Contact( #BR09wAlm3.%X9 )
   END_RUNG wire#w1
   // the same network as SCL:
   "BMS1".BR09xAlmSt := #BR09wAlm1.%X0 OR #BR09wAlm1.%X1 OR #BR09wAlm1.%X2 OR #BR09wAlm1.%X3 OR #BR09wAlm1.%X4 OR #BR09wAlm1.%X5 OR #BR09wAlm1.%X6 OR #BR09wAlm1.%X7 OR #BR09wAlm1.%X8 OR #BR09wAlm1.%X9 OR #BR09wAlm1.%X10 OR #BR09wAlm1.%X11 OR #BR09wAlm1.%X12 OR #BR09wAlm1.%X13 OR #BR09wAlm3.%X0 OR #BR09wAlm3.%X8 OR #BR09wAlm3.%X9;
END_REGION

REGION Network 112: BMS1 BR09 Warning
   RUNG wire#powerrail
      { S7_Templates := "SrcType := Word" } NE_Contact(in1 := #BR09wWarn1, in2 := 0)
      Coil( "BMS1".BR09xWarnSt )
   END_RUNG
   // the same network as SCL:
   "BMS1".BR09xWarnSt := #BR09wWarn1 <> 0;
END_REGION

REGION Network 113: BMS1 BR10 Fault SubSystem
   RUNG wire#powerrail
      Contact( #BR10wAlm2.%X2 )
      Contact( #BR10wAlm2.%X3 )
      wire#w1
      Coil( "BMS1".BR10xSSFltSt )
   END_RUNG
   RUNG wire#powerrail
      Contact( #BR10wAlm3.%X6 )
   END_RUNG wire#w1
   // the same network as SCL:
   "BMS1".BR10xSSFltSt := (#BR10wAlm2.%X2 AND #BR10wAlm2.%X3) OR #BR10wAlm3.%X6;
END_REGION

REGION Network 114: BMS1 BR10 Fault
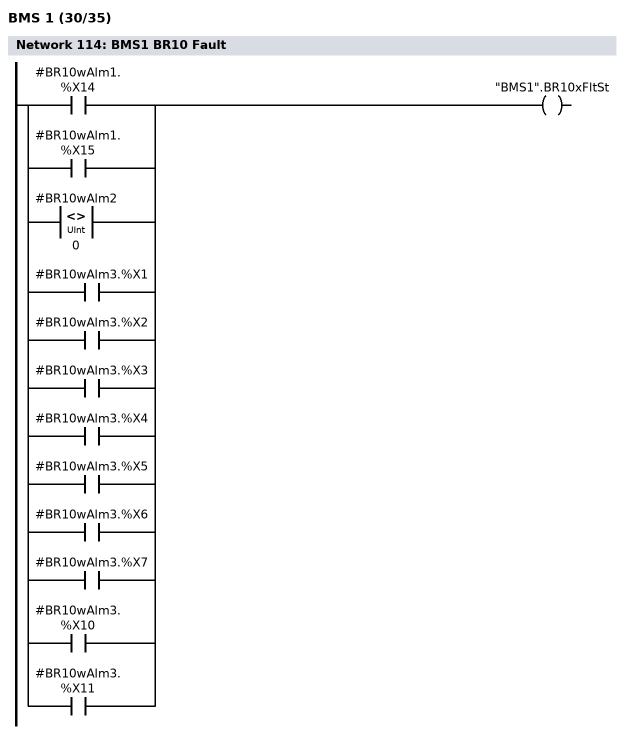
   RUNG wire#powerrail
      Contact( #BR10wAlm1.%X14 )
      wire#w1
      Coil( "BMS1".BR10xFltSt )
   END_RUNG
   RUNG wire#powerrail
      Contact( #BR10wAlm1.%X15 )
   END_RUNG wire#w1
   RUNG wire#powerrail
      { S7_Templates := "SrcType := UInt" } NE_Contact(in1 := #BR10wAlm2, in2 := 0)
   END_RUNG wire#w1
   RUNG wire#powerrail
      Contact( #BR10wAlm3.%X1 )
   END_RUNG wire#w1
   RUNG wire#powerrail
      Contact( #BR10wAlm3.%X2 )
   END_RUNG wire#w1
   RUNG wire#powerrail
      Contact( #BR10wAlm3.%X3 )
   END_RUNG wire#w1
   RUNG wire#powerrail
      Contact( #BR10wAlm3.%X4 )
   END_RUNG wire#w1
   RUNG wire#powerrail
      Contact( #BR10wAlm3.%X5 )
   END_RUNG wire#w1
   RUNG wire#powerrail
      Contact( #BR10wAlm3.%X6 )
   END_RUNG wire#w1
   RUNG wire#powerrail
      Contact( #BR10wAlm3.%X7 )
   END_RUNG wire#w1
   RUNG wire#powerrail
      Contact( #BR10wAlm3.%X10 )
   END_RUNG wire#w1
   RUNG wire#powerrail
      Contact( #BR10wAlm3.%X11 )
   END_RUNG wire#w1
   // the same network as SCL:
   "BMS1".BR10xFltSt := #BR10wAlm1.%X14 OR #BR10wAlm1.%X15 OR (#BR10wAlm2 <> 0) OR #BR10wAlm3.%X1 OR #BR10wAlm3.%X2 OR #BR10wAlm3.%X3 OR #BR10wAlm3.%X4 OR #BR10wAlm3.%X5 OR #BR10wAlm3.%X6 OR #BR10wAlm3.%X7 OR #BR10wAlm3.%X10 OR #BR10wAlm3.%X11;
END_REGION

REGION Network 115: BMS1 BR10 Alarm
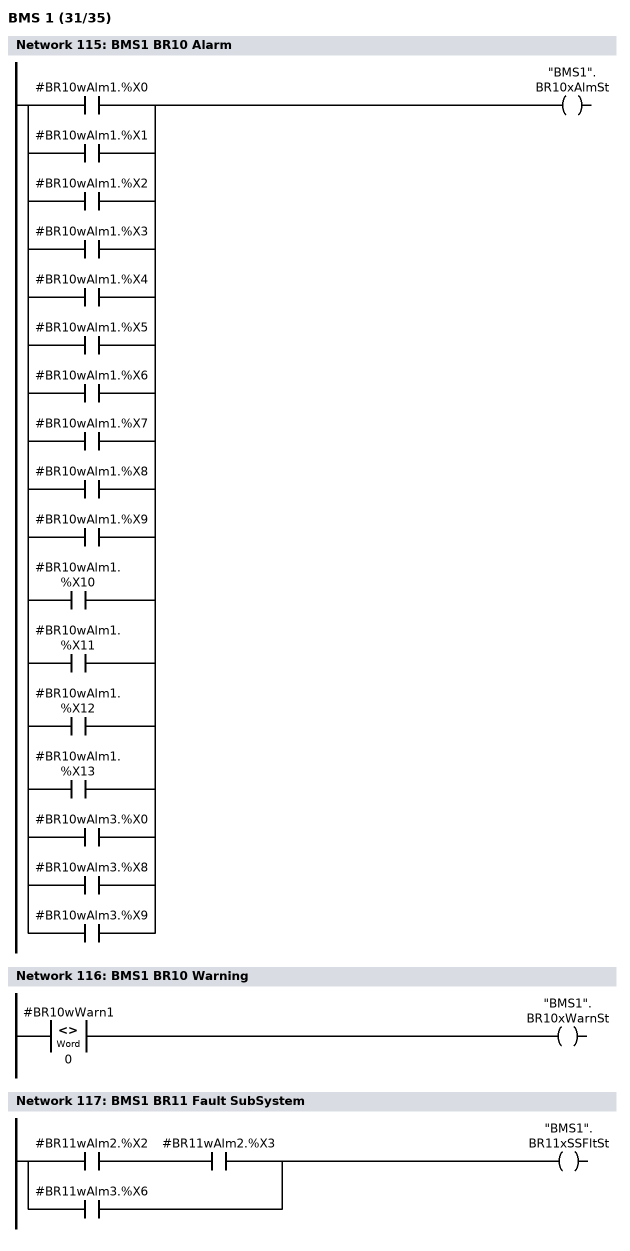
   RUNG wire#powerrail
      Contact( #BR10wAlm1.%X0 )
      wire#w1
      Coil( "BMS1".BR10xAlmSt )
   END_RUNG
   RUNG wire#powerrail
      Contact( #BR10wAlm1.%X1 )
   END_RUNG wire#w1
   RUNG wire#powerrail
      Contact( #BR10wAlm1.%X2 )
   END_RUNG wire#w1
   RUNG wire#powerrail
      Contact( #BR10wAlm1.%X3 )
   END_RUNG wire#w1
   RUNG wire#powerrail
      Contact( #BR10wAlm1.%X4 )
   END_RUNG wire#w1
   RUNG wire#powerrail
      Contact( #BR10wAlm1.%X5 )
   END_RUNG wire#w1
   RUNG wire#powerrail
      Contact( #BR10wAlm1.%X6 )
   END_RUNG wire#w1
   RUNG wire#powerrail
      Contact( #BR10wAlm1.%X7 )
   END_RUNG wire#w1
   RUNG wire#powerrail
      Contact( #BR10wAlm1.%X8 )
   END_RUNG wire#w1
   RUNG wire#powerrail
      Contact( #BR10wAlm1.%X9 )
   END_RUNG wire#w1
   RUNG wire#powerrail
      Contact( #BR10wAlm1.%X10 )
   END_RUNG wire#w1
   RUNG wire#powerrail
      Contact( #BR10wAlm1.%X11 )
   END_RUNG wire#w1
   RUNG wire#powerrail
      Contact( #BR10wAlm1.%X12 )
   END_RUNG wire#w1
   RUNG wire#powerrail
      Contact( #BR10wAlm1.%X13 )
   END_RUNG wire#w1
   RUNG wire#powerrail
      Contact( #BR10wAlm3.%X0 )
   END_RUNG wire#w1
   RUNG wire#powerrail
      Contact( #BR10wAlm3.%X8 )
   END_RUNG wire#w1
   RUNG wire#powerrail
      Contact( #BR10wAlm3.%X9 )
   END_RUNG wire#w1
   // the same network as SCL:
   "BMS1".BR10xAlmSt := #BR10wAlm1.%X0 OR #BR10wAlm1.%X1 OR #BR10wAlm1.%X2 OR #BR10wAlm1.%X3 OR #BR10wAlm1.%X4 OR #BR10wAlm1.%X5 OR #BR10wAlm1.%X6 OR #BR10wAlm1.%X7 OR #BR10wAlm1.%X8 OR #BR10wAlm1.%X9 OR #BR10wAlm1.%X10 OR #BR10wAlm1.%X11 OR #BR10wAlm1.%X12 OR #BR10wAlm1.%X13 OR #BR10wAlm3.%X0 OR #BR10wAlm3.%X8 OR #BR10wAlm3.%X9;
END_REGION

REGION Network 116: BMS1 BR10 Warning
   RUNG wire#powerrail
      { S7_Templates := "SrcType := Word" } NE_Contact(in1 := #BR10wWarn1, in2 := 0)
      Coil( "BMS1".BR10xWarnSt )
   END_RUNG
   // the same network as SCL:
   "BMS1".BR10xWarnSt := #BR10wWarn1 <> 0;
END_REGION

REGION Network 117: BMS1 BR11 Fault SubSystem
   RUNG wire#powerrail
      Contact( #BR11wAlm2.%X2 )
      Contact( #BR11wAlm2.%X3 )
      wire#w1
      Coil( "BMS1".BR11xSSFltSt )
   END_RUNG
   RUNG wire#powerrail
      Contact( #BR11wAlm3.%X6 )
   END_RUNG wire#w1
   // the same network as SCL:
   "BMS1".BR11xSSFltSt := (#BR11wAlm2.%X2 AND #BR11wAlm2.%X3) OR #BR11wAlm3.%X6;
END_REGION

REGION Network 118: BMS1 BR11 Fault
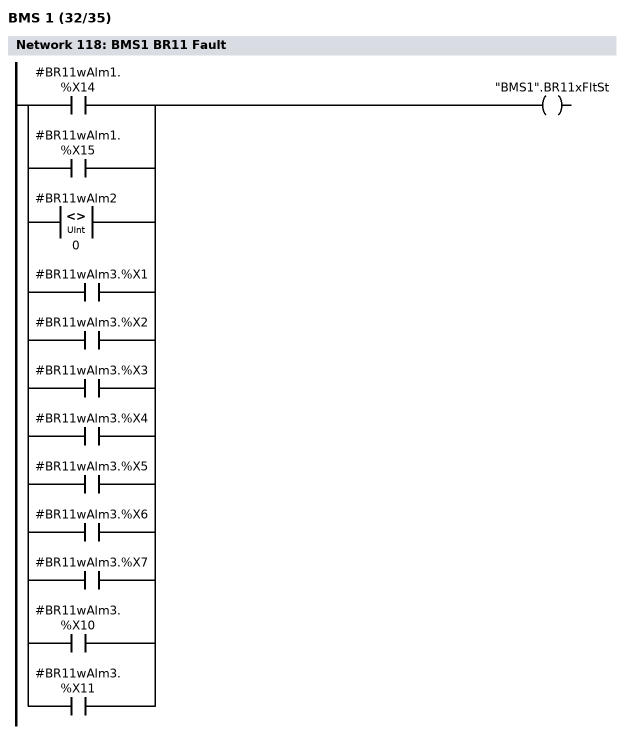
   RUNG wire#powerrail
      Contact( #BR11wAlm1.%X14 )
      wire#w1
      Coil( "BMS1".BR11xFltSt )
   END_RUNG
   RUNG wire#powerrail
      Contact( #BR11wAlm1.%X15 )
   END_RUNG wire#w1
   RUNG wire#powerrail
      { S7_Templates := "SrcType := UInt" } NE_Contact(in1 := #BR11wAlm2, in2 := 0)
   END_RUNG wire#w1
   RUNG wire#powerrail
      Contact( #BR11wAlm3.%X1 )
   END_RUNG wire#w1
   RUNG wire#powerrail
      Contact( #BR11wAlm3.%X2 )
   END_RUNG wire#w1
   RUNG wire#powerrail
      Contact( #BR11wAlm3.%X3 )
   END_RUNG wire#w1
   RUNG wire#powerrail
      Contact( #BR11wAlm3.%X4 )
   END_RUNG wire#w1
   RUNG wire#powerrail
      Contact( #BR11wAlm3.%X5 )
   END_RUNG wire#w1
   RUNG wire#powerrail
      Contact( #BR11wAlm3.%X6 )
   END_RUNG wire#w1
   RUNG wire#powerrail
      Contact( #BR11wAlm3.%X7 )
   END_RUNG wire#w1
   RUNG wire#powerrail
      Contact( #BR11wAlm3.%X10 )
   END_RUNG wire#w1
   RUNG wire#powerrail
      Contact( #BR11wAlm3.%X11 )
   END_RUNG wire#w1
   // the same network as SCL:
   "BMS1".BR11xFltSt := #BR11wAlm1.%X14 OR #BR11wAlm1.%X15 OR (#BR11wAlm2 <> 0) OR #BR11wAlm3.%X1 OR #BR11wAlm3.%X2 OR #BR11wAlm3.%X3 OR #BR11wAlm3.%X4 OR #BR11wAlm3.%X5 OR #BR11wAlm3.%X6 OR #BR11wAlm3.%X7 OR #BR11wAlm3.%X10 OR #BR11wAlm3.%X11;
END_REGION

REGION Network 119: BMS1 BR11 Alarm
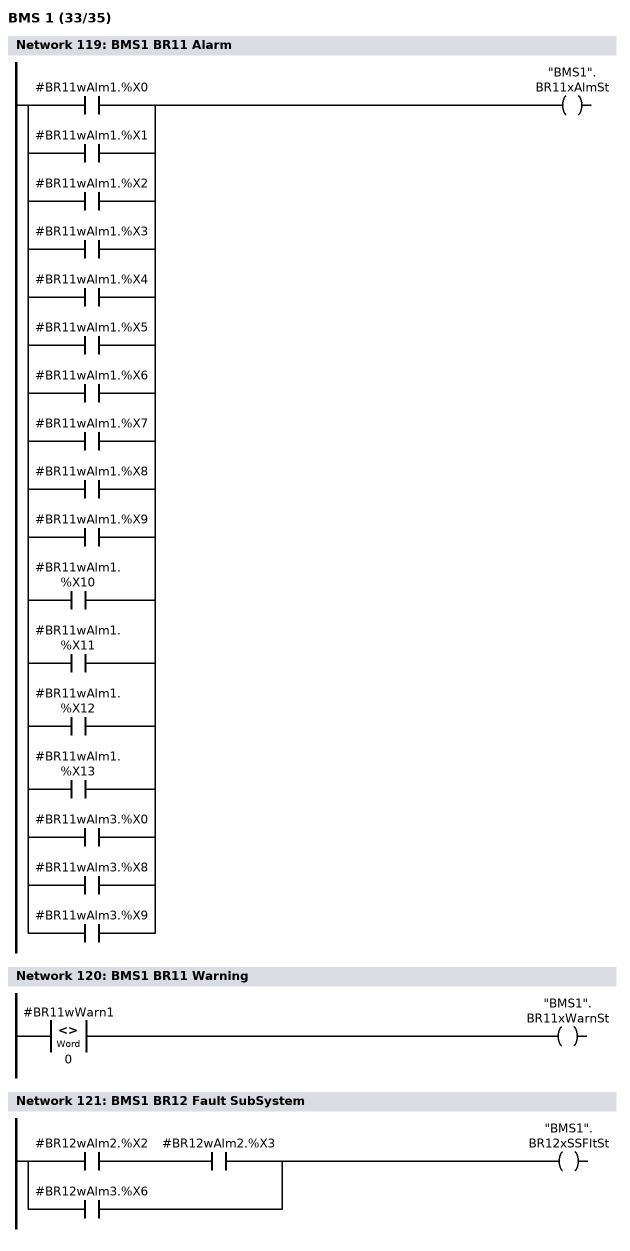
   RUNG wire#powerrail
      Contact( #BR11wAlm1.%X0 )
      wire#w1
      Coil( "BMS1".BR11xAlmSt )
   END_RUNG
   RUNG wire#powerrail
      Contact( #BR11wAlm1.%X1 )
   END_RUNG wire#w1
   RUNG wire#powerrail
      Contact( #BR11wAlm1.%X2 )
   END_RUNG wire#w1
   RUNG wire#powerrail
      Contact( #BR11wAlm1.%X3 )
   END_RUNG wire#w1
   RUNG wire#powerrail
      Contact( #BR11wAlm1.%X4 )
   END_RUNG wire#w1
   RUNG wire#powerrail
      Contact( #BR11wAlm1.%X5 )
   END_RUNG wire#w1
   RUNG wire#powerrail
      Contact( #BR11wAlm1.%X6 )
   END_RUNG wire#w1
   RUNG wire#powerrail
      Contact( #BR11wAlm1.%X7 )
   END_RUNG wire#w1
   RUNG wire#powerrail
      Contact( #BR11wAlm1.%X8 )
   END_RUNG wire#w1
   RUNG wire#powerrail
      Contact( #BR11wAlm1.%X9 )
   END_RUNG wire#w1
   RUNG wire#powerrail
      Contact( #BR11wAlm1.%X10 )
   END_RUNG wire#w1
   RUNG wire#powerrail
      Contact( #BR11wAlm1.%X11 )
   END_RUNG wire#w1
   RUNG wire#powerrail
      Contact( #BR11wAlm1.%X12 )
   END_RUNG wire#w1
   RUNG wire#powerrail
      Contact( #BR11wAlm1.%X13 )
   END_RUNG wire#w1
   RUNG wire#powerrail
      Contact( #BR11wAlm3.%X0 )
   END_RUNG wire#w1
   RUNG wire#powerrail
      Contact( #BR11wAlm3.%X8 )
   END_RUNG wire#w1
   RUNG wire#powerrail
      Contact( #BR11wAlm3.%X9 )
   END_RUNG wire#w1
   // the same network as SCL:
   "BMS1".BR11xAlmSt := #BR11wAlm1.%X0 OR #BR11wAlm1.%X1 OR #BR11wAlm1.%X2 OR #BR11wAlm1.%X3 OR #BR11wAlm1.%X4 OR #BR11wAlm1.%X5 OR #BR11wAlm1.%X6 OR #BR11wAlm1.%X7 OR #BR11wAlm1.%X8 OR #BR11wAlm1.%X9 OR #BR11wAlm1.%X10 OR #BR11wAlm1.%X11 OR #BR11wAlm1.%X12 OR #BR11wAlm1.%X13 OR #BR11wAlm3.%X0 OR #BR11wAlm3.%X8 OR #BR11wAlm3.%X9;
END_REGION

REGION Network 120: BMS1 BR11 Warning
   RUNG wire#powerrail
      { S7_Templates := "SrcType := Word" } NE_Contact(in1 := #BR11wWarn1, in2 := 0)
      Coil( "BMS1".BR11xWarnSt )
   END_RUNG
   // the same network as SCL:
   "BMS1".BR11xWarnSt := #BR11wWarn1 <> 0;
END_REGION

REGION Network 121: BMS1 BR12 Fault SubSystem
   RUNG wire#powerrail
      Contact( #BR12wAlm2.%X2 )
      Contact( #BR12wAlm2.%X3 )
      wire#w1
      Coil( "BMS1".BR12xSSFltSt )
   END_RUNG
   RUNG wire#powerrail
      Contact( #BR12wAlm3.%X6 )
   END_RUNG wire#w1
   // the same network as SCL:
   "BMS1".BR12xSSFltSt := (#BR12wAlm2.%X2 AND #BR12wAlm2.%X3) OR #BR12wAlm3.%X6;
END_REGION

REGION Network 122: BMS1 BR12 Fault
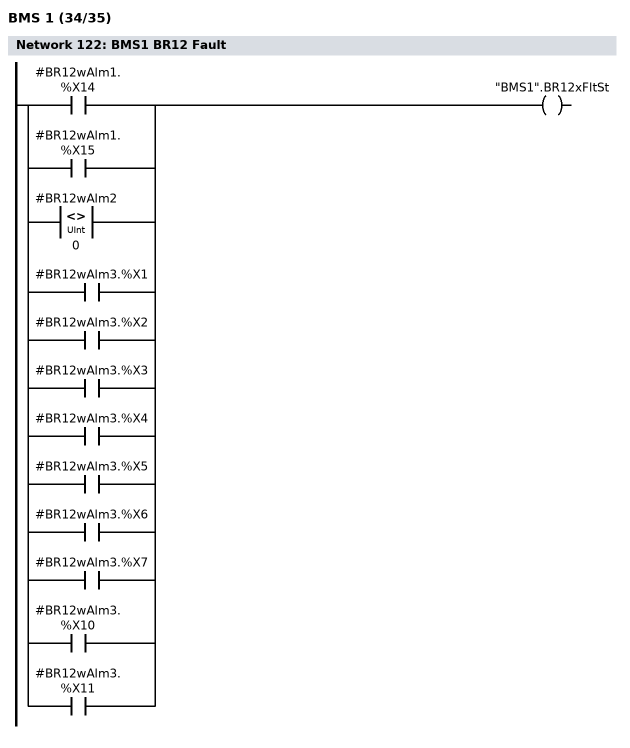
   RUNG wire#powerrail
      Contact( #BR12wAlm1.%X14 )
      wire#w1
      Coil( "BMS1".BR12xFltSt )
   END_RUNG
   RUNG wire#powerrail
      Contact( #BR12wAlm1.%X15 )
   END_RUNG wire#w1
   RUNG wire#powerrail
      { S7_Templates := "SrcType := UInt" } NE_Contact(in1 := #BR12wAlm2, in2 := 0)
   END_RUNG wire#w1
   RUNG wire#powerrail
      Contact( #BR12wAlm3.%X1 )
   END_RUNG wire#w1
   RUNG wire#powerrail
      Contact( #BR12wAlm3.%X2 )
   END_RUNG wire#w1
   RUNG wire#powerrail
      Contact( #BR12wAlm3.%X3 )
   END_RUNG wire#w1
   RUNG wire#powerrail
      Contact( #BR12wAlm3.%X4 )
   END_RUNG wire#w1
   RUNG wire#powerrail
      Contact( #BR12wAlm3.%X5 )
   END_RUNG wire#w1
   RUNG wire#powerrail
      Contact( #BR12wAlm3.%X6 )
   END_RUNG wire#w1
   RUNG wire#powerrail
      Contact( #BR12wAlm3.%X7 )
   END_RUNG wire#w1
   RUNG wire#powerrail
      Contact( #BR12wAlm3.%X10 )
   END_RUNG wire#w1
   RUNG wire#powerrail
      Contact( #BR12wAlm3.%X11 )
   END_RUNG wire#w1
   // the same network as SCL:
   "BMS1".BR12xFltSt := #BR12wAlm1.%X14 OR #BR12wAlm1.%X15 OR (#BR12wAlm2 <> 0) OR #BR12wAlm3.%X1 OR #BR12wAlm3.%X2 OR #BR12wAlm3.%X3 OR #BR12wAlm3.%X4 OR #BR12wAlm3.%X5 OR #BR12wAlm3.%X6 OR #BR12wAlm3.%X7 OR #BR12wAlm3.%X10 OR #BR12wAlm3.%X11;
END_REGION

REGION Network 123: BMS1 BR12 Alarm
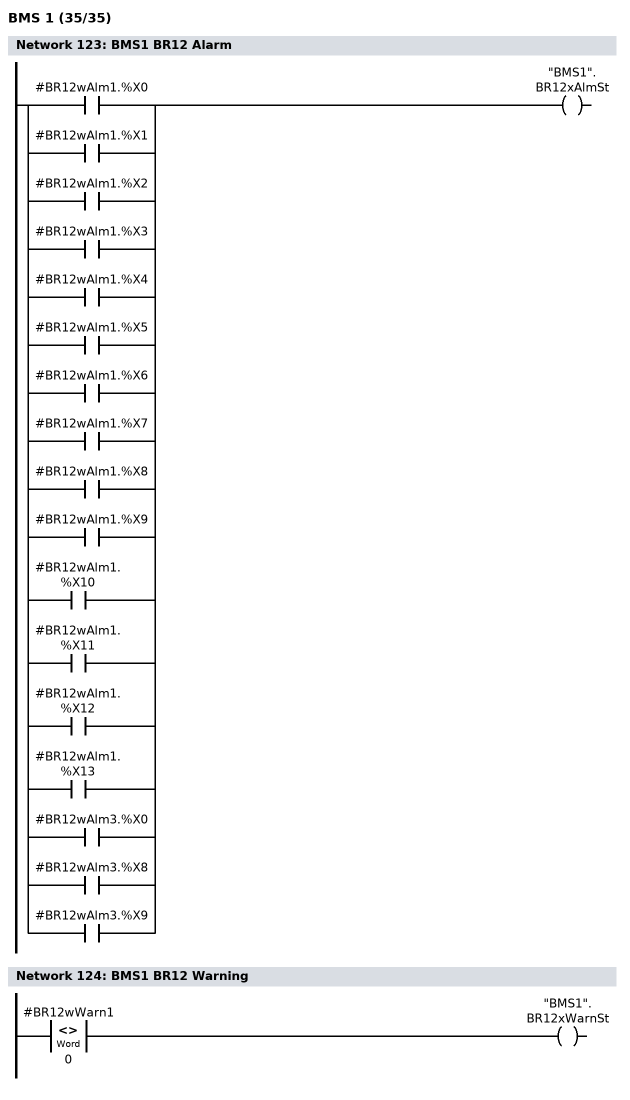
   RUNG wire#powerrail
      Contact( #BR12wAlm1.%X0 )
      wire#w1
      Coil( "BMS1".BR12xAlmSt )
   END_RUNG
   RUNG wire#powerrail
      Contact( #BR12wAlm1.%X1 )
   END_RUNG wire#w1
   RUNG wire#powerrail
      Contact( #BR12wAlm1.%X2 )
   END_RUNG wire#w1
   RUNG wire#powerrail
      Contact( #BR12wAlm1.%X3 )
   END_RUNG wire#w1
   RUNG wire#powerrail
      Contact( #BR12wAlm1.%X4 )
   END_RUNG wire#w1
   RUNG wire#powerrail
      Contact( #BR12wAlm1.%X5 )
   END_RUNG wire#w1
   RUNG wire#powerrail
      Contact( #BR12wAlm1.%X6 )
   END_RUNG wire#w1
   RUNG wire#powerrail
      Contact( #BR12wAlm1.%X7 )
   END_RUNG wire#w1
   RUNG wire#powerrail
      Contact( #BR12wAlm1.%X8 )
   END_RUNG wire#w1
   RUNG wire#powerrail
      Contact( #BR12wAlm1.%X9 )
   END_RUNG wire#w1
   RUNG wire#powerrail
      Contact( #BR12wAlm1.%X10 )
   END_RUNG wire#w1
   RUNG wire#powerrail
      Contact( #BR12wAlm1.%X11 )
   END_RUNG wire#w1
   RUNG wire#powerrail
      Contact( #BR12wAlm1.%X12 )
   END_RUNG wire#w1
   RUNG wire#powerrail
      Contact( #BR12wAlm1.%X13 )
   END_RUNG wire#w1
   RUNG wire#powerrail
      Contact( #BR12wAlm3.%X0 )
   END_RUNG wire#w1
   RUNG wire#powerrail
      Contact( #BR12wAlm3.%X8 )
   END_RUNG wire#w1
   RUNG wire#powerrail
      Contact( #BR12wAlm3.%X9 )
   END_RUNG wire#w1
   // the same network as SCL:
   "BMS1".BR12xAlmSt := #BR12wAlm1.%X0 OR #BR12wAlm1.%X1 OR #BR12wAlm1.%X2 OR #BR12wAlm1.%X3 OR #BR12wAlm1.%X4 OR #BR12wAlm1.%X5 OR #BR12wAlm1.%X6 OR #BR12wAlm1.%X7 OR #BR12wAlm1.%X8 OR #BR12wAlm1.%X9 OR #BR12wAlm1.%X10 OR #BR12wAlm1.%X11 OR #BR12wAlm1.%X12 OR #BR12wAlm1.%X13 OR #BR12wAlm3.%X0 OR #BR12wAlm3.%X8 OR #BR12wAlm3.%X9;
END_REGION

REGION Network 124: BMS1 BR12 Warning
   RUNG wire#powerrail
      { S7_Templates := "SrcType := Word" } NE_Contact(in1 := #BR12wWarn1, in2 := 0)
      Coil( "BMS1".BR12xWarnSt )
   END_RUNG
   // the same network as SCL:
   "BMS1".BR12xWarnSt := #BR12wWarn1 <> 0;
END_REGION
END_FUNCTION

FUNCTION "BMS 2 (F)" : Void   // FC22, LAD
TITLE = ModBus TCP for CATL Battery
{ S7_Optimized_Access := 'TRUE' }
VERSION : 0.1
// stored: AutoNumber false, IsIECCheckEnabled false, SetENOAutomatically false, UDAEnableTagReadback false
   VAR_TEMP
      xSpare : Bool;
      BBwAlm1 : Word;
      BBwWarn1 : Word;
      BR01wAlm1 : Word;
      BR01wAlm2 : Word;
      BR01wAlm3 : Word;
      BR01wWarn1 : Word;
      BR02wAlm1 : Word;
      BR02wAlm2 : Word;
      BR02wAlm3 : Word;
      BR02wWarn1 : Word;
      BR03wAlm1 : Word;
      BR03wAlm2 : Word;
      BR03wAlm3 : Word;
      BR03wWarn1 : Word;
      BR04wAlm1 : Word;
      BR04wAlm2 : Word;
      BR04wAlm3 : Word;
      BR04wWarn1 : Word;
      BR05wAlm1 : Word;
      BR05wAlm2 : Word;
      BR05wAlm3 : Word;
      BR05wWarn1 : Word;
      BR06wAlm1 : Word;
      BR06wAlm2 : Word;
      BR06wAlm3 : Word;
      BR06wWarn1 : Word;
      BR07wAlm1 : Word;
      BR07wAlm2 : Word;
      BR07wAlm3 : Word;
      BR07wWarn1 : Word;
      BR08wAlm1 : Word;
      BR08wAlm2 : Word;
      BR08wAlm3 : Word;
      BR08wWarn1 : Word;
      BR09wAlm1 : Word;
      BR09wAlm2 : Word;
      BR09wAlm3 : Word;
      BR09wWarn1 : Word;
      BR10wAlm1 : Word;
      BR10wAlm2 : Word;
      BR10wAlm3 : Word;
      BR10wWarn1 : Word;
   END_VAR
BEGIN

REGION Network 1: Function Modbus Client
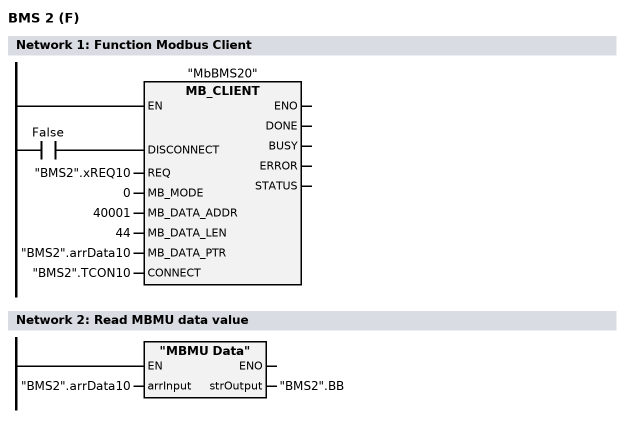
   RUNG wire#powerrail
      "MbBMS20".MB_CLIENT(DISCONNECT := wire#w1, REQ := "BMS2".xREQ10, MB_MODE := 0, MB_DATA_ADDR := 40001, MB_DATA_LEN := 44, MB_DATA_PTR := "BMS2".arrData10, CONNECT := "BMS2".TCON10, DONE =>, BUSY =>, ERROR =>, STATUS =>)
   END_RUNG
   RUNG wire#powerrail
      Contact( False )
   END_RUNG wire#w1
   // the same network as SCL:
   "MbBMS20"(DISCONNECT := False,   // MB_CLIENT
             REQ := "BMS2".xREQ10,
             MB_MODE := 0,
             MB_DATA_ADDR := 40001,
             MB_DATA_LEN := 44,
             MB_DATA_PTR := "BMS2".arrData10,
             CONNECT := "BMS2".TCON10);
END_REGION

REGION Network 2: Read MBMU data value
   RUNG wire#powerrail
      "MBMU Data"(arrInput := "BMS2".arrData10, strOutput => "BMS2".BB)
   END_RUNG
   // the same network as SCL:
   "MBMU Data"(arrInput := "BMS2".arrData10, strOutput => "BMS2".BB);
END_REGION
END_FUNCTION

FUNCTION "BMS 2 (M)" : Void   // FC24, LAD
TITLE = ModBus TCP for CATL Battery
{ S7_Optimized_Access := 'TRUE' }
VERSION : 0.1
// stored: AutoNumber false, IsIECCheckEnabled false, SetENOAutomatically false, UDAEnableTagReadback false
   VAR_TEMP
      xSpare : Bool;
      BBwAlm1 : Word;
      BBwWarn1 : Word;
      BR01wAlm1 : Word;
      BR01wAlm2 : Word;
      BR01wAlm3 : Word;
      BR01wWarn1 : Word;
      BR02wAlm1 : Word;
      BR02wAlm2 : Word;
      BR02wAlm3 : Word;
      BR02wWarn1 : Word;
      BR03wAlm1 : Word;
      BR03wAlm2 : Word;
      BR03wAlm3 : Word;
      BR03wWarn1 : Word;
      BR04wAlm1 : Word;
      BR04wAlm2 : Word;
      BR04wAlm3 : Word;
      BR04wWarn1 : Word;
      BR05wAlm1 : Word;
      BR05wAlm2 : Word;
      BR05wAlm3 : Word;
      BR05wWarn1 : Word;
      BR06wAlm1 : Word;
      BR06wAlm2 : Word;
      BR06wAlm3 : Word;
      BR06wWarn1 : Word;
      BR07wAlm1 : Word;
      BR07wAlm2 : Word;
      BR07wAlm3 : Word;
      BR07wWarn1 : Word;
      BR08wAlm1 : Word;
      BR08wAlm2 : Word;
      BR08wAlm3 : Word;
      BR08wWarn1 : Word;
      BR09wAlm1 : Word;
      BR09wAlm2 : Word;
      BR09wAlm3 : Word;
      BR09wWarn1 : Word;
      BR10wAlm1 : Word;
      BR10wAlm2 : Word;
      BR10wAlm3 : Word;
      BR10wWarn1 : Word;
   END_VAR
BEGIN

REGION Network 1: Function Modbus Client
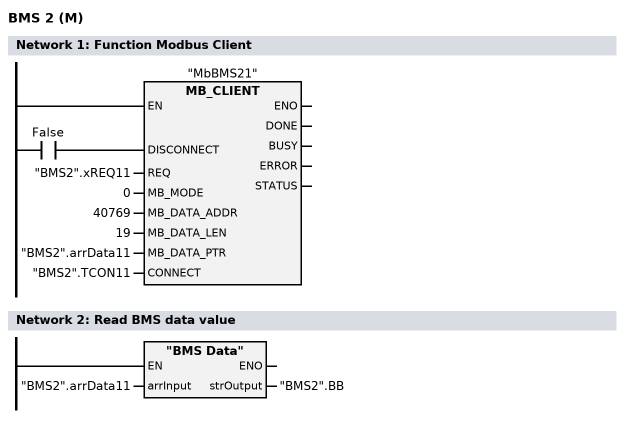
   RUNG wire#powerrail
      "MbBMS21".MB_CLIENT(DISCONNECT := wire#w1, REQ := "BMS2".xREQ11, MB_MODE := 0, MB_DATA_ADDR := 40769, MB_DATA_LEN := 19, MB_DATA_PTR := "BMS2".arrData11, CONNECT := "BMS2".TCON11, DONE =>, BUSY =>, ERROR =>, STATUS =>)
   END_RUNG
   RUNG wire#powerrail
      Contact( False )
   END_RUNG wire#w1
   // the same network as SCL:
   "MbBMS21"(DISCONNECT := False,   // MB_CLIENT
             REQ := "BMS2".xREQ11,
             MB_MODE := 0,
             MB_DATA_ADDR := 40769,
             MB_DATA_LEN := 19,
             MB_DATA_PTR := "BMS2".arrData11,
             CONNECT := "BMS2".TCON11);
END_REGION

REGION Network 2: Read BMS data value
   RUNG wire#powerrail
      "BMS Data"(arrInput := "BMS2".arrData11, strOutput => "BMS2".BB)
   END_RUNG
   // the same network as SCL:
   "BMS Data"(arrInput := "BMS2".arrData11, strOutput => "BMS2".BB);
END_REGION
END_FUNCTION

FUNCTION "BMS 2 (S)" : Void   // FC26, LAD
TITLE = ModBus TCP for CATL Battery
{ S7_Optimized_Access := 'TRUE' }
VERSION : 0.1
// stored: AutoNumber false, IsIECCheckEnabled false, SetENOAutomatically false, UDAEnableTagReadback false
   VAR_TEMP
      xSpare : Bool;
      BBwAlm1 : Word;
      BBwWarn1 : Word;
      BR01wAlm1 : Word;
      BR01wAlm2 : Word;
      BR01wAlm3 : Word;
      BR01wWarn1 : Word;
      BR02wAlm1 : Word;
      BR02wAlm2 : Word;
      BR02wAlm3 : Word;
      BR02wWarn1 : Word;
      BR03wAlm1 : Word;
      BR03wAlm2 : Word;
      BR03wAlm3 : Word;
      BR03wWarn1 : Word;
      BR04wAlm1 : Word;
      BR04wAlm2 : Word;
      BR04wAlm3 : Word;
      BR04wWarn1 : Word;
      BR05wAlm1 : Word;
      BR05wAlm2 : Word;
      BR05wAlm3 : Word;
      BR05wWarn1 : Word;
      BR06wAlm1 : Word;
      BR06wAlm2 : Word;
      BR06wAlm3 : Word;
      BR06wWarn1 : Word;
      BR07wAlm1 : Word;
      BR07wAlm2 : Word;
      BR07wAlm3 : Word;
      BR07wWarn1 : Word;
      BR08wAlm1 : Word;
      BR08wAlm2 : Word;
      BR08wAlm3 : Word;
      BR08wWarn1 : Word;
      BR09wAlm1 : Word;
      BR09wAlm2 : Word;
      BR09wAlm3 : Word;
      BR09wWarn1 : Word;
      BR10wAlm1 : Word;
      BR10wAlm2 : Word;
      BR10wAlm3 : Word;
      BR10wWarn1 : Word;
   END_VAR
   VAR_TEMP   // added for the SCL form of the ladder/FBD networks
      _w1 : Bool;
   END_VAR
BEGIN

REGION Network 1: Function Modbus Client
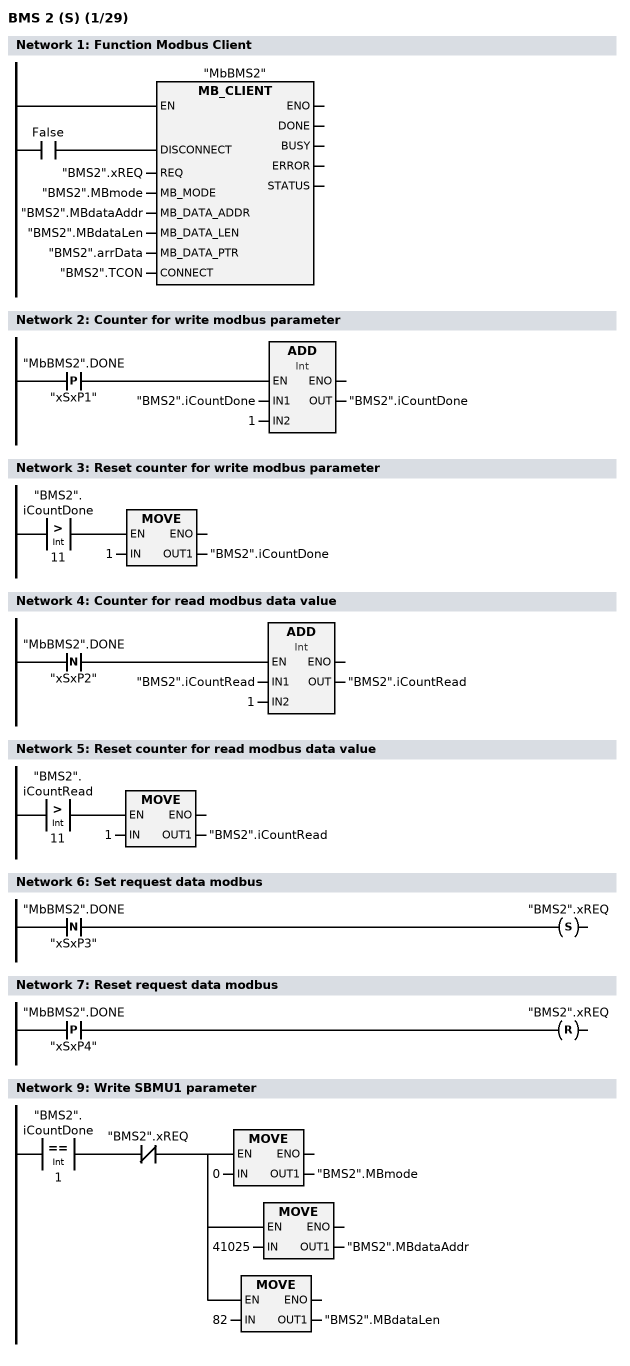
   RUNG wire#powerrail
      "MbBMS2".MB_CLIENT(DISCONNECT := wire#w1, REQ := "BMS2".xREQ, MB_MODE := "BMS2".MBmode, MB_DATA_ADDR := "BMS2".MBdataAddr, MB_DATA_LEN := "BMS2".MBdataLen, MB_DATA_PTR := "BMS2".arrData, CONNECT := "BMS2".TCON, DONE =>, BUSY =>, ERROR =>, STATUS =>)
   END_RUNG
   RUNG wire#powerrail
      Contact( False )
   END_RUNG wire#w1
   // the same network as SCL:
   "MbBMS2"(DISCONNECT := False,   // MB_CLIENT
            REQ := "BMS2".xREQ,
            MB_MODE := "BMS2".MBmode,
            MB_DATA_ADDR := "BMS2".MBdataAddr,
            MB_DATA_LEN := "BMS2".MBdataLen,
            MB_DATA_PTR := "BMS2".arrData,
            CONNECT := "BMS2".TCON);
END_REGION

REGION Network 2: Counter for write modbus parameter
   RUNG wire#powerrail
      P_Contact(operand := "MbBMS2".DONE, bit := "xSxP1")
      { S7_Templates := "SrcType := Int" } Add(in1 := "BMS2".iCountDone, in2 := 1, out => "BMS2".iCountDone)
   END_RUNG
   // the same network as SCL:
   #_w1 := "MbBMS2".DONE AND NOT "xSxP1";   // rising edge of "MbBMS2".DONE
   "xSxP1" := "MbBMS2".DONE;
   IF #_w1 THEN "BMS2".iCountDone := "BMS2".iCountDone + 1; END_IF;
END_REGION

REGION Network 3: Reset counter for write modbus parameter
   RUNG wire#powerrail
      { S7_Templates := "SrcType := Int" } GT_Contact(in1 := "BMS2".iCountDone, in2 := 11)
      Move(in := 1, out1 => "BMS2".iCountDone)
   END_RUNG
   // the same network as SCL:
   IF "BMS2".iCountDone > 11 THEN "BMS2".iCountDone := 1; END_IF;
END_REGION

REGION Network 4: Counter for read modbus data value
   RUNG wire#powerrail
      N_Contact(operand := "MbBMS2".DONE, bit := "xSxP2")
      { S7_Templates := "SrcType := Int" } Add(in1 := "BMS2".iCountRead, in2 := 1, out => "BMS2".iCountRead)
   END_RUNG
   // the same network as SCL:
   #_w1 := NOT "MbBMS2".DONE AND "xSxP2";   // falling edge of "MbBMS2".DONE
   "xSxP2" := "MbBMS2".DONE;
   IF #_w1 THEN "BMS2".iCountRead := "BMS2".iCountRead + 1; END_IF;
END_REGION

REGION Network 5: Reset counter for read modbus data value
   RUNG wire#powerrail
      { S7_Templates := "SrcType := Int" } GT_Contact(in1 := "BMS2".iCountRead, in2 := 11)
      Move(in := 1, out1 => "BMS2".iCountRead)
   END_RUNG
   // the same network as SCL:
   IF "BMS2".iCountRead > 11 THEN "BMS2".iCountRead := 1; END_IF;
END_REGION

REGION Network 6: Set request data modbus
   RUNG wire#powerrail
      N_Contact(operand := "MbBMS2".DONE, bit := "xSxP3")
      S_Coil( "BMS2".xREQ )
   END_RUNG
   // the same network as SCL:
   #_w1 := NOT "MbBMS2".DONE AND "xSxP3";   // falling edge of "MbBMS2".DONE
   "xSxP3" := "MbBMS2".DONE;
   IF #_w1 THEN "BMS2".xREQ := TRUE; END_IF;
END_REGION

REGION Network 7: Reset request data modbus
   RUNG wire#powerrail
      P_Contact(operand := "MbBMS2".DONE, bit := "xSxP4")
      R_Coil( "BMS2".xREQ )
   END_RUNG
   // the same network as SCL:
   #_w1 := "MbBMS2".DONE AND NOT "xSxP4";   // rising edge of "MbBMS2".DONE
   "xSxP4" := "MbBMS2".DONE;
   IF #_w1 THEN "BMS2".xREQ := FALSE; END_IF;
END_REGION

REGION Network 9: Write SBMU1 parameter
   RUNG wire#powerrail
      { S7_Templates := "SrcType := Int" } EQ_Contact(in1 := "BMS2".iCountDone, in2 := 1)
      I_Contact( "BMS2".xREQ )
      wire#w1
      Move(in := 0, out1 => "BMS2".MBmode)
   END_RUNG
   RUNG wire#w1
      Move(in := 41025, out1 => "BMS2".MBdataAddr)
   END_RUNG
   RUNG wire#w1
      Move(in := 82, out1 => "BMS2".MBdataLen)
   END_RUNG
   // the same network as SCL:
   IF ("BMS2".iCountDone = 1) AND NOT "BMS2".xREQ THEN
       "BMS2".MBmode := 0;
       "BMS2".MBdataAddr := 41025;
       "BMS2".MBdataLen := 82;
   END_IF;
END_REGION

REGION Network 10: Read SBMU1 data value
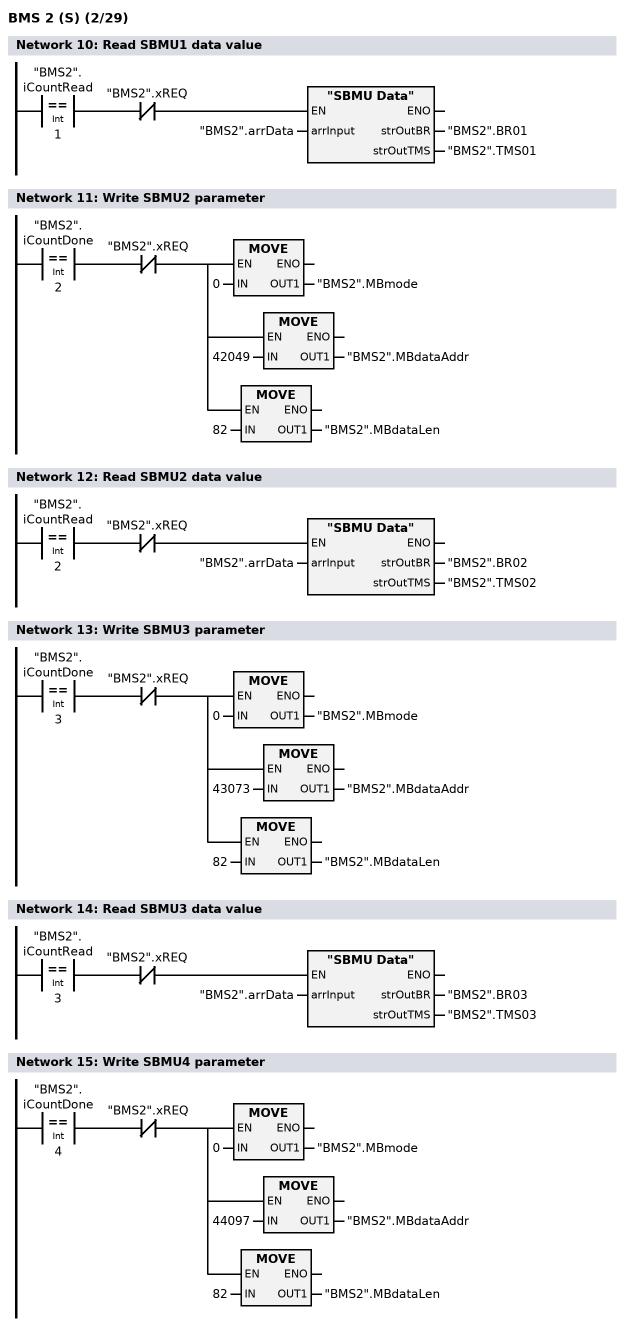
   RUNG wire#powerrail
      { S7_Templates := "SrcType := Int" } EQ_Contact(in1 := "BMS2".iCountRead, in2 := 1)
      I_Contact( "BMS2".xREQ )
      "SBMU Data"(arrInput := "BMS2".arrData, strOutBR => "BMS2".BR01, strOutTMS => "BMS2".TMS01)
   END_RUNG
   // the same network as SCL:
   IF ("BMS2".iCountRead = 1) AND NOT "BMS2".xREQ THEN
       "SBMU Data"(arrInput := "BMS2".arrData, strOutBR => "BMS2".BR01, strOutTMS => "BMS2".TMS01);
   END_IF;
END_REGION

REGION Network 11: Write SBMU2 parameter
   RUNG wire#powerrail
      { S7_Templates := "SrcType := Int" } EQ_Contact(in1 := "BMS2".iCountDone, in2 := 2)
      I_Contact( "BMS2".xREQ )
      wire#w1
      Move(in := 0, out1 => "BMS2".MBmode)
   END_RUNG
   RUNG wire#w1
      Move(in := 42049, out1 => "BMS2".MBdataAddr)
   END_RUNG
   RUNG wire#w1
      Move(in := 82, out1 => "BMS2".MBdataLen)
   END_RUNG
   // the same network as SCL:
   IF ("BMS2".iCountDone = 2) AND NOT "BMS2".xREQ THEN
       "BMS2".MBmode := 0;
       "BMS2".MBdataAddr := 42049;
       "BMS2".MBdataLen := 82;
   END_IF;
END_REGION

REGION Network 12: Read SBMU2 data value
   RUNG wire#powerrail
      { S7_Templates := "SrcType := Int" } EQ_Contact(in1 := "BMS2".iCountRead, in2 := 2)
      I_Contact( "BMS2".xREQ )
      "SBMU Data"(arrInput := "BMS2".arrData, strOutBR => "BMS2".BR02, strOutTMS => "BMS2".TMS02)
   END_RUNG
   // the same network as SCL:
   IF ("BMS2".iCountRead = 2) AND NOT "BMS2".xREQ THEN
       "SBMU Data"(arrInput := "BMS2".arrData, strOutBR => "BMS2".BR02, strOutTMS => "BMS2".TMS02);
   END_IF;
END_REGION

REGION Network 13: Write SBMU3 parameter
   RUNG wire#powerrail
      { S7_Templates := "SrcType := Int" } EQ_Contact(in1 := "BMS2".iCountDone, in2 := 3)
      I_Contact( "BMS2".xREQ )
      wire#w1
      Move(in := 0, out1 => "BMS2".MBmode)
   END_RUNG
   RUNG wire#w1
      Move(in := 43073, out1 => "BMS2".MBdataAddr)
   END_RUNG
   RUNG wire#w1
      Move(in := 82, out1 => "BMS2".MBdataLen)
   END_RUNG
   // the same network as SCL:
   IF ("BMS2".iCountDone = 3) AND NOT "BMS2".xREQ THEN
       "BMS2".MBmode := 0;
       "BMS2".MBdataAddr := 43073;
       "BMS2".MBdataLen := 82;
   END_IF;
END_REGION

REGION Network 14: Read SBMU3 data value
   RUNG wire#powerrail
      { S7_Templates := "SrcType := Int" } EQ_Contact(in1 := "BMS2".iCountRead, in2 := 3)
      I_Contact( "BMS2".xREQ )
      "SBMU Data"(arrInput := "BMS2".arrData, strOutBR => "BMS2".BR03, strOutTMS => "BMS2".TMS03)
   END_RUNG
   // the same network as SCL:
   IF ("BMS2".iCountRead = 3) AND NOT "BMS2".xREQ THEN
       "SBMU Data"(arrInput := "BMS2".arrData, strOutBR => "BMS2".BR03, strOutTMS => "BMS2".TMS03);
   END_IF;
END_REGION

REGION Network 15: Write SBMU4 parameter
   RUNG wire#powerrail
      { S7_Templates := "SrcType := Int" } EQ_Contact(in1 := "BMS2".iCountDone, in2 := 4)
      I_Contact( "BMS2".xREQ )
      wire#w1
      Move(in := 0, out1 => "BMS2".MBmode)
   END_RUNG
   RUNG wire#w1
      Move(in := 44097, out1 => "BMS2".MBdataAddr)
   END_RUNG
   RUNG wire#w1
      Move(in := 82, out1 => "BMS2".MBdataLen)
   END_RUNG
   // the same network as SCL:
   IF ("BMS2".iCountDone = 4) AND NOT "BMS2".xREQ THEN
       "BMS2".MBmode := 0;
       "BMS2".MBdataAddr := 44097;
       "BMS2".MBdataLen := 82;
   END_IF;
END_REGION

REGION Network 16: Read SBMU4 data value
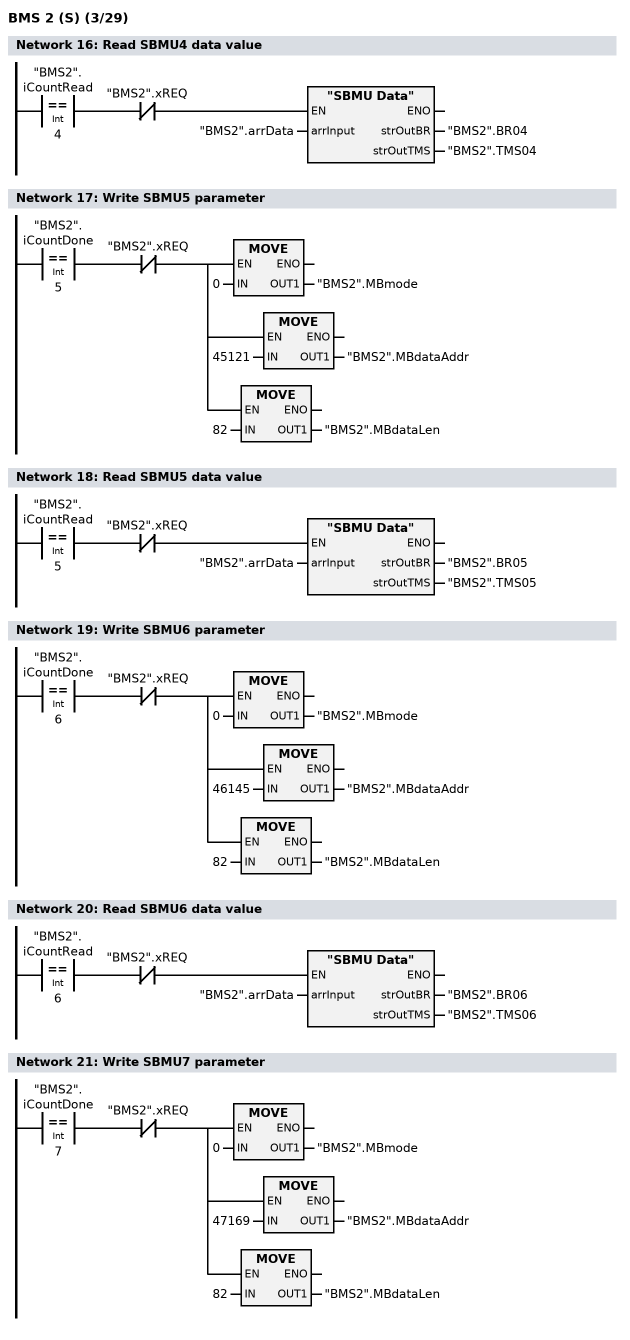
   RUNG wire#powerrail
      { S7_Templates := "SrcType := Int" } EQ_Contact(in1 := "BMS2".iCountRead, in2 := 4)
      I_Contact( "BMS2".xREQ )
      "SBMU Data"(arrInput := "BMS2".arrData, strOutBR => "BMS2".BR04, strOutTMS => "BMS2".TMS04)
   END_RUNG
   // the same network as SCL:
   IF ("BMS2".iCountRead = 4) AND NOT "BMS2".xREQ THEN
       "SBMU Data"(arrInput := "BMS2".arrData, strOutBR => "BMS2".BR04, strOutTMS => "BMS2".TMS04);
   END_IF;
END_REGION

REGION Network 17: Write SBMU5 parameter
   RUNG wire#powerrail
      { S7_Templates := "SrcType := Int" } EQ_Contact(in1 := "BMS2".iCountDone, in2 := 5)
      I_Contact( "BMS2".xREQ )
      wire#w1
      Move(in := 0, out1 => "BMS2".MBmode)
   END_RUNG
   RUNG wire#w1
      Move(in := 45121, out1 => "BMS2".MBdataAddr)
   END_RUNG
   RUNG wire#w1
      Move(in := 82, out1 => "BMS2".MBdataLen)
   END_RUNG
   // the same network as SCL:
   IF ("BMS2".iCountDone = 5) AND NOT "BMS2".xREQ THEN
       "BMS2".MBmode := 0;
       "BMS2".MBdataAddr := 45121;
       "BMS2".MBdataLen := 82;
   END_IF;
END_REGION

REGION Network 18: Read SBMU5 data value
   RUNG wire#powerrail
      { S7_Templates := "SrcType := Int" } EQ_Contact(in1 := "BMS2".iCountRead, in2 := 5)
      I_Contact( "BMS2".xREQ )
      "SBMU Data"(arrInput := "BMS2".arrData, strOutBR => "BMS2".BR05, strOutTMS => "BMS2".TMS05)
   END_RUNG
   // the same network as SCL:
   IF ("BMS2".iCountRead = 5) AND NOT "BMS2".xREQ THEN
       "SBMU Data"(arrInput := "BMS2".arrData, strOutBR => "BMS2".BR05, strOutTMS => "BMS2".TMS05);
   END_IF;
END_REGION

REGION Network 19: Write SBMU6 parameter
   RUNG wire#powerrail
      { S7_Templates := "SrcType := Int" } EQ_Contact(in1 := "BMS2".iCountDone, in2 := 6)
      I_Contact( "BMS2".xREQ )
      wire#w1
      Move(in := 0, out1 => "BMS2".MBmode)
   END_RUNG
   RUNG wire#w1
      Move(in := 46145, out1 => "BMS2".MBdataAddr)
   END_RUNG
   RUNG wire#w1
      Move(in := 82, out1 => "BMS2".MBdataLen)
   END_RUNG
   // the same network as SCL:
   IF ("BMS2".iCountDone = 6) AND NOT "BMS2".xREQ THEN
       "BMS2".MBmode := 0;
       "BMS2".MBdataAddr := 46145;
       "BMS2".MBdataLen := 82;
   END_IF;
END_REGION

REGION Network 20: Read SBMU6 data value
   RUNG wire#powerrail
      { S7_Templates := "SrcType := Int" } EQ_Contact(in1 := "BMS2".iCountRead, in2 := 6)
      I_Contact( "BMS2".xREQ )
      "SBMU Data"(arrInput := "BMS2".arrData, strOutBR => "BMS2".BR06, strOutTMS => "BMS2".TMS06)
   END_RUNG
   // the same network as SCL:
   IF ("BMS2".iCountRead = 6) AND NOT "BMS2".xREQ THEN
       "SBMU Data"(arrInput := "BMS2".arrData, strOutBR => "BMS2".BR06, strOutTMS => "BMS2".TMS06);
   END_IF;
END_REGION

REGION Network 21: Write SBMU7 parameter
   RUNG wire#powerrail
      { S7_Templates := "SrcType := Int" } EQ_Contact(in1 := "BMS2".iCountDone, in2 := 7)
      I_Contact( "BMS2".xREQ )
      wire#w1
      Move(in := 0, out1 => "BMS2".MBmode)
   END_RUNG
   RUNG wire#w1
      Move(in := 47169, out1 => "BMS2".MBdataAddr)
   END_RUNG
   RUNG wire#w1
      Move(in := 82, out1 => "BMS2".MBdataLen)
   END_RUNG
   // the same network as SCL:
   IF ("BMS2".iCountDone = 7) AND NOT "BMS2".xREQ THEN
       "BMS2".MBmode := 0;
       "BMS2".MBdataAddr := 47169;
       "BMS2".MBdataLen := 82;
   END_IF;
END_REGION

REGION Network 22: Read SBMU7 data value
